SPLINE
SPL {X  -145.877, Y  +737.201, Z    +0.000, E1  +394.468, E3 -267040.191}
SPL {X  -152.550, Y  +719.721, Z    +0.000, E1  +387.728, E3 -267055.680}
SPL {X  -157.145, Y  +701.536, Z    +0.000, E1  +379.368, E3 -267065.135}
SPL {X  -159.035, Y  +688.952, Z    +0.000, E1  +372.676, E3 -267069.176}
SPL {X  -159.756, Y  +680.154, Z    +0.000, E1  +367.520, E3 -267070.903}
SPL {X  -159.986, Y  +672.560, Z    +0.000, E1  +362.636, E3 -267071.801}
SPL {X  -159.990, Y  +668.344, Z    +0.000, E1  +359.382, E3 -267072.067}
SPL {X  -159.990, Y  +664.070, Z    +0.000, E1  +354.975, E3 -267072.395}
SPL {X  -159.990, Y  +656.953, Z    +0.000, E1  +346.040, E3 -267073.462}
SPL {X  -159.990, Y  +644.589, Z    +0.000, E1  +330.989, E3 -267076.873}
SPL {X  -159.990, Y  +605.095, Z    +0.000, E1  +310.486, E3 -267101.964}
SPL {X  -159.990, Y  +546.155, Z    +0.000, E1  +305.539, E3 -267164.723}
SPL {X  -159.990, Y  +539.348, Z    +0.000, E1  +305.531, E3 -267175.026}
SPL {X  -159.990, Y  +530.752, Z    +0.000, E1  +305.518, E3 -267188.034}
SPL {X  -159.990, Y  +522.797, Z    +0.000, E1  +305.537, E3 -267200.117}
SPL {X  -159.990, Y  +515.332, Z    +0.000, E1  +305.526, E3 -267211.406}
SPL {X  -159.990, Y  +508.047, Z    +0.000, E1  +305.531, E3 -267222.422}
SPL {X  -159.990, Y  +501.296, Z    +0.000, E1  +305.518, E3 -267232.644}
SPL {X  -159.990, Y  +487.558, Z    +0.000, E1  +304.151, E3 -267244.274}
SPL {X  -159.990, Y  +454.926, Z    +0.000, E1  +299.433, E3 -267255.714}
SPL {X  -159.990, Y  +449.697, Z    +0.000, E1  +300.191, E3 -267267.176}
SPL {X  -159.990, Y  +445.847, Z    +0.000, E1  +300.905, E3 -267276.799}
SPL {X  -159.990, Y  +439.266, Z    +0.000, E1  +301.568, E3 -267289.882}
SPL {X  -159.990, Y  +432.883, Z    +0.000, E1  +302.386, E3 -267303.573}
SPL {X  -159.990, Y  +429.044, Z    +0.000, E1  +303.109, E3 -267313.463}
SPL {X  -159.990, Y  +425.222, Z    +0.000, E1  +304.101, E3 -267325.360}
SPL {X  -159.990, Y  +418.562, Z    +0.000, E1  +304.950, E3 -267340.518}
SPL {X  -159.990, Y  +407.911, Z    +0.000, E1  +305.062, E3 -267357.109}
SPL {X  -159.990, Y  +400.284, Z    +0.000, E1  +305.103, E3 -267368.543}
SPL {X  -159.990, Y  +391.119, Z    +0.000, E1  +305.052, E3 -267382.131}
SPL {X  -159.988, Y  +381.720, Z    +0.000, E1  +305.103, E3 -267396.239}
SPL {X  -159.786, Y  +374.425, Z    +0.000, E1  +305.121, E3 -267407.287}
SPL {X  -159.015, Y  +364.863, Z    +0.000, E1  +305.220, E3 -267422.303}
SPL {X  -157.966, Y  +357.131, Z    +0.000, E1  +305.441, E3 -267434.993}
SPL {X  -156.775, Y  +350.586, Z    +0.000, E1  +305.627, E3 -267445.967}
SPL {X  -155.027, Y  +342.959, Z    +0.000, E1  +305.926, E3 -267459.140}
SPL {X  -152.882, Y  +335.340, Z    +0.000, E1  +306.305, E3 -267472.683}
SPL {X  -150.681, Y  +328.723, Z    +0.000, E1  +306.710, E3 -267484.777}
SPL {X  -148.661, Y  +323.366, Z    +0.000, E1  +307.100, E3 -267494.786}
SPL {X  -147.089, Y  +319.560, Z    +0.000, E1  +307.396, E3 -267502.002}
SPL {X  -145.161, Y  +315.232, Z    +0.000, E1  +307.745, E3 -267510.282}
SPL {X  -142.534, Y  +309.830, Z    +0.000, E1  +308.237, E3 -267520.787}
SPL {X  -132.342, Y  +292.599, Z    +0.000, E1  +315.826, E3 -267618.075}
ENDSPLINE

SPLINE
SPL {X  -151.238, Y  +330.309, Z    +0.000, E1  +330.693, E3 -267691.232}
SPL {X  -156.949, Y  +351.453, Z    +0.000, E1  +340.161, E3 -267703.393}
SPL {X  -159.024, Y  +364.945, Z    +0.000, E1  +347.297, E3 -267707.811}
SPL {X  -159.758, Y  +373.891, Z    +0.000, E1  +352.513, E3 -267709.699}
SPL {X  -159.985, Y  +381.208, Z    +0.000, E1  +357.184, E3 -267710.582}
SPL {X  -159.990, Y  +384.493, Z    +0.000, E1  +359.676, E3 -267710.807}
SPL {X  -159.990, Y  +387.327, Z    +0.000, E1  +362.137, E3 -267710.990}
SPL {X  -159.990, Y  +392.053, Z    +0.000, E1  +367.477, E3 -267711.454}
SPL {X  -159.990, Y  +396.158, Z    +0.000, E1  +372.775, E3 -267712.080}
SPL {X  -159.990, Y  +401.377, Z    +0.000, E1  +379.398, E3 -267713.260}
SPL {X  -159.990, Y  +411.365, Z    +0.000, E1  +390.630, E3 -267716.469}
SPL {X  -159.990, Y  +450.467, Z    +0.000, E1  +410.183, E3 -267740.118}
SPL {X  -159.990, Y  +509.934, Z    +0.000, E1  +414.923, E3 -267802.736}
SPL {X  -159.990, Y  +516.848, Z    +0.000, E1  +414.930, E3 -267813.025}
SPL {X  -159.990, Y  +524.818, Z    +0.000, E1  +414.933, E3 -267824.896}
SPL {X  -159.990, Y  +532.100, Z    +0.000, E1  +414.924, E3 -267835.749}
SPL {X  -159.990, Y  +539.391, Z    +0.000, E1  +414.933, E3 -267846.601}
SPL {X  -159.990, Y  +546.283, Z    +0.000, E1  +414.924, E3 -267856.873}
SPL {X  -159.990, Y  +553.734, Z    +0.000, E1  +414.938, E3 -267867.960}
SPL {X  -159.990, Y  +564.956, Z    +0.000, E1  +414.973, E3 -267884.631}
SPL {X  -159.990, Y  +577.902, Z    +0.000, E1  +414.969, E3 -267903.921}
SPL {X  -159.990, Y  +588.063, Z    +0.000, E1  +414.931, E3 -267919.112}
SPL {X  -159.990, Y  +595.273, Z    +0.000, E1  +414.928, E3 -267929.835}
SPL {X  -159.990, Y  +602.326, Z    +0.000, E1  +414.932, E3 -267940.336}
SPL {X  -159.990, Y  +609.708, Z    +0.000, E1  +414.930, E3 -267951.342}
SPL {X  -159.990, Y  +618.088, Z    +0.000, E1  +414.948, E3 -267963.771}
SPL {X  -159.990, Y  +625.928, Z    +0.000, E1  +414.931, E3 -267975.467}
SPL {X  -159.990, Y  +632.991, Z    +0.000, E1  +414.938, E3 -267985.970}
SPL {X  -159.990, Y  +639.033, Z    +0.000, E1  +414.931, E3 -267994.978}
SPL {X  -159.990, Y  +646.303, Z    +0.000, E1  +414.946, E3 -268005.766}
SPL {X  -159.990, Y  +656.335, Z    +0.000, E1  +414.969, E3 -268020.668}
SPL {X  -159.990, Y  +664.577, Z    +0.000, E1  +414.924, E3 -268033.045}
SPL {X  -159.989, Y  +672.128, Z    +0.000, E1  +414.946, E3 -268044.262}
SPL {X  -159.636, Y  +682.136, Z    +0.000, E1  +414.901, E3 -268059.520}
SPL {X  -158.805, Y  +690.934, Z    +0.000, E1  +414.742, E3 -268073.531}
SPL {X  -157.890, Y  +697.337, Z    +0.000, E1  +414.571, E3 -268084.052}
SPL {X  -156.492, Y  +704.774, Z    +0.000, E1  +414.365, E3 -268096.531}
SPL {X  -154.917, Y  +711.470, Z    +0.000, E1  +414.052, E3 -268108.191}
SPL {X  -153.204, Y  +717.603, Z    +0.000, E1  +413.775, E3 -268119.037}
SPL {X  -151.355, Y  +723.351, Z    +0.000, E1  +413.415, E3 -268129.508}
SPL {X  -148.967, Y  +729.859, Z    +0.000, E1  +413.026, E3 -268141.520}
SPL {X  -145.862, Y  +737.236, Z    +0.000, E1  +412.427, E3 -268155.575}
SPL {X  -142.777, Y  +743.691, Z    +0.000, E1  +411.831, E3 -268168.118}
SPL {X  -132.301, Y  +761.463, Z    +0.000, E1  +405.510, E3 -268247.403}
ENDSPLINE

SPLINE
SPL {X  -145.877, Y  +737.201, Z    +0.000, E1  +394.468, E3 -268330.514}
SPL {X  -152.550, Y  +719.721, Z    +0.000, E1  +387.728, E3 -268346.003}
SPL {X  -157.145, Y  +701.536, Z    +0.000, E1  +379.368, E3 -268355.458}
SPL {X  -159.035, Y  +688.952, Z    +0.000, E1  +372.676, E3 -268359.499}
SPL {X  -159.756, Y  +680.154, Z    +0.000, E1  +367.520, E3 -268361.225}
SPL {X  -159.986, Y  +672.560, Z    +0.000, E1  +362.636, E3 -268362.123}
SPL {X  -159.990, Y  +668.344, Z    +0.000, E1  +359.382, E3 -268362.389}
SPL {X  -159.990, Y  +664.070, Z    +0.000, E1  +354.975, E3 -268362.718}
SPL {X  -159.990, Y  +656.953, Z    +0.000, E1  +346.040, E3 -268363.784}
SPL {X  -159.990, Y  +644.589, Z    +0.000, E1  +330.989, E3 -268367.196}
SPL {X  -159.990, Y  +605.095, Z    +0.000, E1  +310.486, E3 -268392.287}
SPL {X  -159.990, Y  +546.155, Z    +0.000, E1  +305.539, E3 -268455.045}
SPL {X  -159.990, Y  +539.348, Z    +0.000, E1  +305.531, E3 -268465.349}
SPL {X  -159.990, Y  +530.752, Z    +0.000, E1  +305.518, E3 -268478.356}
SPL {X  -159.990, Y  +522.797, Z    +0.000, E1  +305.537, E3 -268490.439}
SPL {X  -159.990, Y  +515.332, Z    +0.000, E1  +305.526, E3 -268501.728}
SPL {X  -159.990, Y  +508.047, Z    +0.000, E1  +305.531, E3 -268512.745}
SPL {X  -159.990, Y  +501.296, Z    +0.000, E1  +305.518, E3 -268522.966}
SPL {X  -159.990, Y  +487.558, Z    +0.000, E1  +304.151, E3 -268534.597}
SPL {X  -159.990, Y  +454.926, Z    +0.000, E1  +299.433, E3 -268546.036}
SPL {X  -159.990, Y  +449.697, Z    +0.000, E1  +300.191, E3 -268557.499}
SPL {X  -159.990, Y  +445.847, Z    +0.000, E1  +300.905, E3 -268567.122}
SPL {X  -159.990, Y  +439.266, Z    +0.000, E1  +301.568, E3 -268580.205}
SPL {X  -159.990, Y  +432.883, Z    +0.000, E1  +302.386, E3 -268593.895}
SPL {X  -159.990, Y  +428.299, Z    +0.000, E1  +303.316, E3 -268606.299}
SPL {X  -159.990, Y  +424.402, Z    +0.000, E1  +304.297, E3 -268617.974}
SPL {X  -159.990, Y  +420.083, Z    +0.000, E1  +304.918, E3 -268628.258}
SPL {X  -159.990, Y  +412.567, Z    +0.000, E1  +305.072, E3 -268640.482}
SPL {X  -159.990, Y  +405.235, Z    +0.000, E1  +305.098, E3 -268651.471}
SPL {X  -159.990, Y  +400.284, Z    +0.000, E1  +305.103, E3 -268658.865}
SPL {X  -159.990, Y  +391.119, Z    +0.000, E1  +305.052, E3 -268672.454}
SPL {X  -159.988, Y  +381.720, Z    +0.000, E1  +305.103, E3 -268686.561}
SPL {X  -159.786, Y  +374.425, Z    +0.000, E1  +305.121, E3 -268697.609}
SPL {X  -159.015, Y  +364.863, Z    +0.000, E1  +305.220, E3 -268712.626}
SPL {X  -157.966, Y  +357.131, Z    +0.000, E1  +305.441, E3 -268725.316}
SPL {X  -156.775, Y  +350.586, Z    +0.000, E1  +305.627, E3 -268736.290}
SPL {X  -155.397, Y  +344.442, Z    +0.000, E1  +305.886, E3 -268746.906}
SPL {X  -153.976, Y  +339.046, Z    +0.000, E1  +306.128, E3 -268756.398}
SPL {X  -152.417, Y  +333.859, Z    +0.000, E1  +306.416, E3 -268765.724}
SPL {X  -150.681, Y  +328.723, Z    +0.000, E1  +306.710, E3 -268775.100}
SPL {X  -147.884, Y  +321.449, Z    +0.000, E1  +307.200, E3 -268788.673}
SPL {X  -144.518, Y  +313.862, Z    +0.000, E1  +307.832, E3 -268803.219}
SPL {X  -141.812, Y  +308.430, Z    +0.000, E1  +308.410, E3 -268813.906}
SPL {X  -132.342, Y  +292.599, Z    +0.000, E1  +315.826, E3 -268908.398}
ENDSPLINE

SPLINE
SPL {X  -151.238, Y  +330.309, Z    +0.000, E1  +330.693, E3 -268981.554}
SPL {X  -156.949, Y  +351.453, Z    +0.000, E1  +340.161, E3 -268993.715}
SPL {X  -159.024, Y  +364.945, Z    +0.000, E1  +347.297, E3 -268998.133}
SPL {X  -159.878, Y  +376.512, Z    +0.000, E1  +354.071, E3 -269000.385}
SPL {X  -159.990, Y  +382.403, Z    +0.000, E1  +358.090, E3 -269001.004}
SPL {X  -159.990, Y  +385.261, Z    +0.000, E1  +360.259, E3 -269001.175}
SPL {X  -159.990, Y  +389.002, Z    +0.000, E1  +363.890, E3 -269001.453}
SPL {X  -159.990, Y  +394.493, Z    +0.000, E1  +370.512, E3 -269002.128}
SPL {X  -159.990, Y  +401.377, Z    +0.000, E1  +379.398, E3 -269003.583}
SPL {X  -159.990, Y  +411.365, Z    +0.000, E1  +390.630, E3 -269006.791}
SPL {X  -159.990, Y  +450.467, Z    +0.000, E1  +410.183, E3 -269030.440}
SPL {X  -159.990, Y  +509.934, Z    +0.000, E1  +414.923, E3 -269093.059}
SPL {X  -159.990, Y  +516.848, Z    +0.000, E1  +414.930, E3 -269103.347}
SPL {X  -159.990, Y  +524.818, Z    +0.000, E1  +414.933, E3 -269115.219}
SPL {X  -159.990, Y  +532.100, Z    +0.000, E1  +414.924, E3 -269126.072}
SPL {X  -159.990, Y  +539.391, Z    +0.000, E1  +414.933, E3 -269136.924}
SPL {X  -159.990, Y  +546.283, Z    +0.000, E1  +414.924, E3 -269147.196}
SPL {X  -159.990, Y  +553.734, Z    +0.000, E1  +414.938, E3 -269158.282}
SPL {X  -159.990, Y  +564.956, Z    +0.000, E1  +414.973, E3 -269174.954}
SPL {X  -159.990, Y  +577.902, Z    +0.000, E1  +414.969, E3 -269194.243}
SPL {X  -159.990, Y  +588.063, Z    +0.000, E1  +414.931, E3 -269209.434}
SPL {X  -159.990, Y  +595.273, Z    +0.000, E1  +414.928, E3 -269220.158}
SPL {X  -159.990, Y  +602.326, Z    +0.000, E1  +414.932, E3 -269230.658}
SPL {X  -159.990, Y  +609.708, Z    +0.000, E1  +414.930, E3 -269241.665}
SPL {X  -159.990, Y  +618.088, Z    +0.000, E1  +414.948, E3 -269254.094}
SPL {X  -159.990, Y  +625.928, Z    +0.000, E1  +414.931, E3 -269265.790}
SPL {X  -159.990, Y  +635.803, Z    +0.000, E1  +414.980, E3 -269280.418}
SPL {X  -159.990, Y  +646.303, Z    +0.000, E1  +414.946, E3 -269296.088}
SPL {X  -159.990, Y  +653.312, Z    +0.000, E1  +414.932, E3 -269306.540}
SPL {X  -159.990, Y  +658.943, Z    +0.000, E1  +414.931, E3 -269314.938}
SPL {X  -159.990, Y  +667.151, Z    +0.000, E1  +414.954, E3 -269327.157}
SPL {X  -159.885, Y  +677.285, Z    +0.000, E1  +414.936, E3 -269342.352}
SPL {X  -159.482, Y  +684.244, Z    +0.000, E1  +414.840, E3 -269353.204}
SPL {X  -158.805, Y  +690.934, Z    +0.000, E1  +414.742, E3 -269363.853}
SPL {X  -157.890, Y  +697.337, Z    +0.000, E1  +414.571, E3 -269374.375}
SPL {X  -156.492, Y  +704.774, Z    +0.000, E1  +414.365, E3 -269386.854}
SPL {X  -154.917, Y  +711.470, Z    +0.000, E1  +414.052, E3 -269398.514}
SPL {X  -153.204, Y  +717.603, Z    +0.000, E1  +413.775, E3 -269409.360}
SPL {X  -151.355, Y  +723.351, Z    +0.000, E1  +413.415, E3 -269419.831}
SPL {X  -148.967, Y  +729.859, Z    +0.000, E1  +413.026, E3 -269431.843}
SPL {X  -145.862, Y  +737.236, Z    +0.000, E1  +412.427, E3 -269445.897}
SPL {X  -142.777, Y  +743.691, Z    +0.000, E1  +411.831, E3 -269458.441}
SPL {X  -132.301, Y  +761.463, Z    +0.000, E1  +405.510, E3 -269537.726}
ENDSPLINE

SPLINE
SPL {X  -145.877, Y  +737.201, Z    +0.000, E1  +394.468, E3 -269620.836}
SPL {X  -152.550, Y  +719.721, Z    +0.000, E1  +387.728, E3 -269636.326}
SPL {X  -157.145, Y  +701.536, Z    +0.000, E1  +379.368, E3 -269645.780}
SPL {X  -159.035, Y  +688.952, Z    +0.000, E1  +372.676, E3 -269649.821}
SPL {X  -159.873, Y  +677.622, Z    +0.000, E1  +366.008, E3 -269651.893}
SPL {X  -159.990, Y  +670.381, Z    +0.000, E1  +361.064, E3 -269652.594}
SPL {X  -159.990, Y  +666.603, Z    +0.000, E1  +357.744, E3 -269652.825}
SPL {X  -159.990, Y  +661.750, Z    +0.000, E1  +352.120, E3 -269653.298}
SPL {X  -159.990, Y  +657.656, Z    +0.000, E1  +346.724, E3 -269653.943}
SPL {X  -159.990, Y  +652.023, Z    +0.000, E1  +339.551, E3 -269655.231}
SPL {X  -159.990, Y  +641.935, Z    +0.000, E1  +328.152, E3 -269658.403}
SPL {X  -159.990, Y  +605.095, Z    +0.000, E1  +310.486, E3 -269682.609}
SPL {X  -159.990, Y  +546.155, Z    +0.000, E1  +305.539, E3 -269745.368}
SPL {X  -159.990, Y  +539.348, Z    +0.000, E1  +305.531, E3 -269755.672}
SPL {X  -159.990, Y  +530.752, Z    +0.000, E1  +305.518, E3 -269768.679}
SPL {X  -159.990, Y  +522.797, Z    +0.000, E1  +305.537, E3 -269780.762}
SPL {X  -159.990, Y  +515.332, Z    +0.000, E1  +305.526, E3 -269792.051}
SPL {X  -159.990, Y  +508.047, Z    +0.000, E1  +305.531, E3 -269803.068}
SPL {X  -159.990, Y  +499.403, Z    +0.000, E1  +305.488, E3 -269816.107}
SPL {X  -159.990, Y  +479.413, Z    +0.000, E1  +302.719, E3 -269827.252}
SPL {X  -159.990, Y  +454.926, Z    +0.000, E1  +299.433, E3 -269836.359}
SPL {X  -159.990, Y  +449.697, Z    +0.000, E1  +300.191, E3 -269847.821}
SPL {X  -159.990, Y  +445.847, Z    +0.000, E1  +300.905, E3 -269857.444}
SPL {X  -159.990, Y  +439.266, Z    +0.000, E1  +301.568, E3 -269870.528}
SPL {X  -159.990, Y  +432.883, Z    +0.000, E1  +302.386, E3 -269884.218}
SPL {X  -159.990, Y  +428.299, Z    +0.000, E1  +303.316, E3 -269896.621}
SPL {X  -159.990, Y  +424.402, Z    +0.000, E1  +304.297, E3 -269908.296}
SPL {X  -159.990, Y  +418.562, Z    +0.000, E1  +304.950, E3 -269921.163}
SPL {X  -159.990, Y  +410.722, Z    +0.000, E1  +305.100, E3 -269933.624}
SPL {X  -159.990, Y  +402.790, Z    +0.000, E1  +305.070, E3 -269945.399}
SPL {X  -159.990, Y  +392.953, Z    +0.000, E1  +305.082, E3 -269960.093}
SPL {X  -159.990, Y  +383.354, Z    +0.000, E1  +305.080, E3 -269974.403}
SPL {X  -159.786, Y  +374.425, Z    +0.000, E1  +305.121, E3 -269987.932}
SPL {X  -159.015, Y  +364.863, Z    +0.000, E1  +305.220, E3 -270002.948}
SPL {X  -157.966, Y  +357.131, Z    +0.000, E1  +305.441, E3 -270015.639}
SPL {X  -156.775, Y  +350.586, Z    +0.000, E1  +305.627, E3 -270026.613}
SPL {X  -155.027, Y  +342.959, Z    +0.000, E1  +305.926, E3 -270039.786}
SPL {X  -152.882, Y  +335.340, Z    +0.000, E1  +306.305, E3 -270053.328}
SPL {X  -150.681, Y  +328.723, Z    +0.000, E1  +306.710, E3 -270065.422}
SPL {X  -147.884, Y  +321.449, Z    +0.000, E1  +307.200, E3 -270078.996}
SPL {X  -145.161, Y  +315.232, Z    +0.000, E1  +307.745, E3 -270090.927}
SPL {X  -142.534, Y  +309.830, Z    +0.000, E1  +308.237, E3 -270101.432}
SPL {X  -132.342, Y  +292.599, Z    +0.000, E1  +315.826, E3 -270198.720}
ENDSPLINE

SPLINE
SPL {X  -151.238, Y  +330.309, Z    +0.000, E1  +330.693, E3 -270271.877}
SPL {X  -156.949, Y  +351.453, Z    +0.000, E1  +340.161, E3 -270284.038}
SPL {X  -159.024, Y  +364.945, Z    +0.000, E1  +347.297, E3 -270288.456}
SPL {X  -159.758, Y  +373.891, Z    +0.000, E1  +352.513, E3 -270290.344}
SPL {X  -159.985, Y  +381.208, Z    +0.000, E1  +357.184, E3 -270291.227}
SPL {X  -159.990, Y  +385.261, Z    +0.000, E1  +360.259, E3 -270291.497}
SPL {X  -159.990, Y  +388.094, Z    +0.000, E1  +363.012, E3 -270291.690}
SPL {X  -159.990, Y  +392.053, Z    +0.000, E1  +367.477, E3 -270292.100}
SPL {X  -159.990, Y  +396.158, Z    +0.000, E1  +372.775, E3 -270292.725}
SPL {X  -159.990, Y  +401.377, Z    +0.000, E1  +379.398, E3 -270293.905}
SPL {X  -159.990, Y  +411.365, Z    +0.000, E1  +390.630, E3 -270297.114}
SPL {X  -159.990, Y  +450.467, Z    +0.000, E1  +410.183, E3 -270320.763}
SPL {X  -159.990, Y  +509.934, Z    +0.000, E1  +414.923, E3 -270383.382}
SPL {X  -159.990, Y  +516.848, Z    +0.000, E1  +414.930, E3 -270393.670}
SPL {X  -159.990, Y  +524.818, Z    +0.000, E1  +414.933, E3 -270405.542}
SPL {X  -159.990, Y  +532.100, Z    +0.000, E1  +414.924, E3 -270416.395}
SPL {X  -159.990, Y  +539.391, Z    +0.000, E1  +414.933, E3 -270427.247}
SPL {X  -159.990, Y  +546.283, Z    +0.000, E1  +414.924, E3 -270437.518}
SPL {X  -159.990, Y  +553.734, Z    +0.000, E1  +414.938, E3 -270448.605}
SPL {X  -159.990, Y  +560.657, Z    +0.000, E1  +414.914, E3 -270458.966}
SPL {X  -159.990, Y  +567.311, Z    +0.000, E1  +414.931, E3 -270468.851}
SPL {X  -159.990, Y  +577.902, Z    +0.000, E1  +414.969, E3 -270484.566}
SPL {X  -159.990, Y  +588.063, Z    +0.000, E1  +414.931, E3 -270499.757}
SPL {X  -159.990, Y  +595.273, Z    +0.000, E1  +414.928, E3 -270510.480}
SPL {X  -159.990, Y  +602.326, Z    +0.000, E1  +414.932, E3 -270520.981}
SPL {X  -159.990, Y  +609.708, Z    +0.000, E1  +414.930, E3 -270531.988}
SPL {X  -159.990, Y  +618.088, Z    +0.000, E1  +414.948, E3 -270544.416}
SPL {X  -159.990, Y  +625.928, Z    +0.000, E1  +414.931, E3 -270556.112}
SPL {X  -159.990, Y  +635.803, Z    +0.000, E1  +414.980, E3 -270570.740}
SPL {X  -159.990, Y  +646.303, Z    +0.000, E1  +414.946, E3 -270586.411}
SPL {X  -159.990, Y  +653.312, Z    +0.000, E1  +414.932, E3 -270596.863}
SPL {X  -159.990, Y  +658.943, Z    +0.000, E1  +414.931, E3 -270605.261}
SPL {X  -159.990, Y  +667.151, Z    +0.000, E1  +414.954, E3 -270617.479}
SPL {X  -159.885, Y  +677.285, Z    +0.000, E1  +414.936, E3 -270632.675}
SPL {X  -159.482, Y  +684.244, Z    +0.000, E1  +414.840, E3 -270643.527}
SPL {X  -158.805, Y  +690.934, Z    +0.000, E1  +414.742, E3 -270654.176}
SPL {X  -157.890, Y  +697.337, Z    +0.000, E1  +414.571, E3 -270664.697}
SPL {X  -156.492, Y  +704.774, Z    +0.000, E1  +414.365, E3 -270677.176}
SPL {X  -154.917, Y  +711.470, Z    +0.000, E1  +414.052, E3 -270688.836}
SPL {X  -153.204, Y  +717.603, Z    +0.000, E1  +413.775, E3 -270699.682}
SPL {X  -151.355, Y  +723.351, Z    +0.000, E1  +413.415, E3 -270710.154}
SPL {X  -149.700, Y  +727.952, Z    +0.000, E1  +413.118, E3 -270718.648}
SPL {X  -147.376, Y  +733.767, Z    +0.000, E1  +412.706, E3 -270729.598}
SPL {X  -144.332, Y  +740.529, Z    +0.000, E1  +412.133, E3 -270742.588}
SPL {X  -142.065, Y  +745.081, Z    +0.000, E1  +411.654, E3 -270751.541}
SPL {X  -132.301, Y  +761.463, Z    +0.000, E1  +405.510, E3 -270828.048}
ENDSPLINE

SPLINE
SPL {X  -145.877, Y  +737.201, Z    +0.000, E1  +394.468, E3 -270911.159}
SPL {X  -152.550, Y  +719.721, Z    +0.000, E1  +387.728, E3 -270926.648}
SPL {X  -157.145, Y  +701.536, Z    +0.000, E1  +379.368, E3 -270936.103}
SPL {X  -159.035, Y  +688.952, Z    +0.000, E1  +372.676, E3 -270940.144}
SPL {X  -159.756, Y  +680.154, Z    +0.000, E1  +367.520, E3 -270941.870}
SPL {X  -159.986, Y  +672.560, Z    +0.000, E1  +362.636, E3 -270942.768}
SPL {X  -159.990, Y  +668.344, Z    +0.000, E1  +359.382, E3 -270943.035}
SPL {X  -159.990, Y  +664.070, Z    +0.000, E1  +354.975, E3 -270943.363}
SPL {X  -159.990, Y  +656.953, Z    +0.000, E1  +346.040, E3 -270944.429}
SPL {X  -159.990, Y  +644.589, Z    +0.000, E1  +330.989, E3 -270947.841}
SPL {X  -159.990, Y  +605.095, Z    +0.000, E1  +310.486, E3 -270972.932}
SPL {X  -159.990, Y  +546.155, Z    +0.000, E1  +305.539, E3 -271035.690}
SPL {X  -159.990, Y  +539.348, Z    +0.000, E1  +305.531, E3 -271045.994}
SPL {X  -159.990, Y  +530.752, Z    +0.000, E1  +305.518, E3 -271059.002}
SPL {X  -159.990, Y  +522.797, Z    +0.000, E1  +305.537, E3 -271071.085}
SPL {X  -159.990, Y  +515.332, Z    +0.000, E1  +305.526, E3 -271082.373}
SPL {X  -159.990, Y  +508.047, Z    +0.000, E1  +305.531, E3 -271093.390}
SPL {X  -159.990, Y  +501.296, Z    +0.000, E1  +305.518, E3 -271103.612}
SPL {X  -159.990, Y  +487.558, Z    +0.000, E1  +304.151, E3 -271115.242}
SPL {X  -159.990, Y  +454.926, Z    +0.000, E1  +299.433, E3 -271126.681}
SPL {X  -159.990, Y  +449.697, Z    +0.000, E1  +300.191, E3 -271138.144}
SPL {X  -159.990, Y  +444.026, Z    +0.000, E1  +301.072, E3 -271151.402}
SPL {X  -159.990, Y  +437.596, Z    +0.000, E1  +301.764, E3 -271164.144}
SPL {X  -159.990, Y  +432.883, Z    +0.000, E1  +302.386, E3 -271174.540}
SPL {X  -159.990, Y  +429.044, Z    +0.000, E1  +303.109, E3 -271184.431}
SPL {X  -159.990, Y  +425.222, Z    +0.000, E1  +304.101, E3 -271196.328}
SPL {X  -159.990, Y  +418.562, Z    +0.000, E1  +304.950, E3 -271211.485}
SPL {X  -159.990, Y  +407.911, Z    +0.000, E1  +305.062, E3 -271228.077}
SPL {X  -159.990, Y  +400.284, Z    +0.000, E1  +305.103, E3 -271239.511}
SPL {X  -159.990, Y  +392.953, Z    +0.000, E1  +305.082, E3 -271250.415}
SPL {X  -159.990, Y  +383.354, Z    +0.000, E1  +305.080, E3 -271264.725}
SPL {X  -159.786, Y  +374.425, Z    +0.000, E1  +305.121, E3 -271278.255}
SPL {X  -159.184, Y  +366.462, Z    +0.000, E1  +305.220, E3 -271290.755}
SPL {X  -158.166, Y  +358.413, Z    +0.000, E1  +305.386, E3 -271303.811}
SPL {X  -156.775, Y  +350.586, Z    +0.000, E1  +305.627, E3 -271316.935}
SPL {X  -155.397, Y  +344.442, Z    +0.000, E1  +305.886, E3 -271327.551}
SPL {X  -153.976, Y  +339.046, Z    +0.000, E1  +306.128, E3 -271337.043}
SPL {X  -152.417, Y  +333.859, Z    +0.000, E1  +306.416, E3 -271346.369}
SPL {X  -150.681, Y  +328.723, Z    +0.000, E1  +306.710, E3 -271355.745}
SPL {X  -147.884, Y  +321.449, Z    +0.000, E1  +307.200, E3 -271369.318}
SPL {X  -145.161, Y  +315.232, Z    +0.000, E1  +307.745, E3 -271381.250}
SPL {X  -142.534, Y  +309.830, Z    +0.000, E1  +308.237, E3 -271391.755}
SPL {X  -132.342, Y  +292.599, Z    +0.000, E1  +315.826, E3 -271489.043}
ENDSPLINE

SPLINE
SPL {X  -151.238, Y  +330.309, Z    +0.000, E1  +330.693, E3 -271562.200}
SPL {X  -156.949, Y  +351.453, Z    +0.000, E1  +340.161, E3 -271574.361}
SPL {X  -159.024, Y  +364.945, Z    +0.000, E1  +347.297, E3 -271578.778}
SPL {X  -159.878, Y  +376.512, Z    +0.000, E1  +354.071, E3 -271581.030}
SPL {X  -159.990, Y  +383.659, Z    +0.000, E1  +358.950, E3 -271581.724}
SPL {X  -159.990, Y  +387.327, Z    +0.000, E1  +362.137, E3 -271581.957}
SPL {X  -159.990, Y  +392.053, Z    +0.000, E1  +367.477, E3 -271582.422}
SPL {X  -159.990, Y  +396.158, Z    +0.000, E1  +372.775, E3 -271583.048}
SPL {X  -159.990, Y  +401.377, Z    +0.000, E1  +379.398, E3 -271584.228}
SPL {X  -159.990, Y  +411.365, Z    +0.000, E1  +390.630, E3 -271587.437}
SPL {X  -159.990, Y  +450.467, Z    +0.000, E1  +410.183, E3 -271611.085}
SPL {X  -159.990, Y  +509.934, Z    +0.000, E1  +414.923, E3 -271673.704}
SPL {X  -159.990, Y  +516.848, Z    +0.000, E1  +414.930, E3 -271683.992}
SPL {X  -159.990, Y  +524.818, Z    +0.000, E1  +414.933, E3 -271695.864}
SPL {X  -159.990, Y  +532.100, Z    +0.000, E1  +414.924, E3 -271706.717}
SPL {X  -159.990, Y  +539.391, Z    +0.000, E1  +414.933, E3 -271717.569}
SPL {X  -159.990, Y  +546.283, Z    +0.000, E1  +414.924, E3 -271727.841}
SPL {X  -159.990, Y  +553.734, Z    +0.000, E1  +414.938, E3 -271738.928}
SPL {X  -159.990, Y  +564.956, Z    +0.000, E1  +414.973, E3 -271755.599}
SPL {X  -159.990, Y  +577.902, Z    +0.000, E1  +414.969, E3 -271774.889}
SPL {X  -159.990, Y  +588.063, Z    +0.000, E1  +414.931, E3 -271790.080}
SPL {X  -159.990, Y  +595.273, Z    +0.000, E1  +414.928, E3 -271800.803}
SPL {X  -159.990, Y  +602.326, Z    +0.000, E1  +414.932, E3 -271811.303}
SPL {X  -159.990, Y  +609.708, Z    +0.000, E1  +414.930, E3 -271822.310}
SPL {X  -159.990, Y  +616.306, Z    +0.000, E1  +414.927, E3 -271832.124}
SPL {X  -159.990, Y  +624.320, Z    +0.000, E1  +414.952, E3 -271844.007}
SPL {X  -159.990, Y  +632.991, Z    +0.000, E1  +414.938, E3 -271856.938}
SPL {X  -159.990, Y  +639.033, Z    +0.000, E1  +414.931, E3 -271865.946}
SPL {X  -159.990, Y  +646.303, Z    +0.000, E1  +414.946, E3 -271876.733}
SPL {X  -159.990, Y  +656.335, Z    +0.000, E1  +414.969, E3 -271891.636}
SPL {X  -159.990, Y  +664.577, Z    +0.000, E1  +414.924, E3 -271904.013}
SPL {X  -159.989, Y  +672.128, Z    +0.000, E1  +414.946, E3 -271915.230}
SPL {X  -159.792, Y  +679.466, Z    +0.000, E1  +414.893, E3 -271926.388}
SPL {X  -159.330, Y  +686.016, Z    +0.000, E1  +414.837, E3 -271936.619}
SPL {X  -158.190, Y  +695.432, Z    +0.000, E1  +414.658, E3 -271951.815}
SPL {X  -157.027, Y  +702.151, Z    +0.000, E1  +414.415, E3 -271963.097}
SPL {X  -156.112, Y  +706.513, Z    +0.000, E1  +414.265, E3 -271970.531}
SPL {X  -154.917, Y  +711.470, Z    +0.000, E1  +414.052, E3 -271979.159}
SPL {X  -153.561, Y  +716.398, Z    +0.000, E1  +413.816, E3 -271987.880}
SPL {X  -151.715, Y  +722.287, Z    +0.000, E1  +413.503, E3 -271998.496}
SPL {X  -148.967, Y  +729.859, Z    +0.000, E1  +413.026, E3 -272012.488}
SPL {X  -146.734, Y  +735.264, Z    +0.000, E1  +412.550, E3 -272022.820}
SPL {X  -144.332, Y  +740.529, Z    +0.000, E1  +412.133, E3 -272032.911}
SPL {X  -142.065, Y  +745.081, Z    +0.000, E1  +411.654, E3 -272041.864}
SPL {X  -132.301, Y  +761.463, Z    +0.000, E1  +405.510, E3 -272118.371}
ENDSPLINE

SPLINE
SPL {X  -145.877, Y  +737.201, Z    +0.000, E1  +394.468, E3 -272201.482}
SPL {X  -152.550, Y  +719.721, Z    +0.000, E1  +387.728, E3 -272216.971}
SPL {X  -157.145, Y  +701.536, Z    +0.000, E1  +379.368, E3 -272226.425}
SPL {X  -159.035, Y  +688.952, Z    +0.000, E1  +372.676, E3 -272230.466}
SPL {X  -159.873, Y  +677.622, Z    +0.000, E1  +366.008, E3 -272232.538}
SPL {X  -159.990, Y  +670.381, Z    +0.000, E1  +361.064, E3 -272233.239}
SPL {X  -159.990, Y  +667.647, Z    +0.000, E1  +358.660, E3 -272233.397}
SPL {X  -159.990, Y  +664.070, Z    +0.000, E1  +354.975, E3 -272233.685}
SPL {X  -159.990, Y  +658.737, Z    +0.000, E1  +348.199, E3 -272234.392}
SPL {X  -159.990, Y  +652.023, Z    +0.000, E1  +339.551, E3 -272235.876}
SPL {X  -159.990, Y  +641.935, Z    +0.000, E1  +328.152, E3 -272239.048}
SPL {X  -159.990, Y  +605.095, Z    +0.000, E1  +310.486, E3 -272263.254}
SPL {X  -159.990, Y  +546.155, Z    +0.000, E1  +305.539, E3 -272326.013}
SPL {X  -159.990, Y  +539.348, Z    +0.000, E1  +305.531, E3 -272336.317}
SPL {X  -159.990, Y  +530.752, Z    +0.000, E1  +305.518, E3 -272349.324}
SPL {X  -159.990, Y  +522.797, Z    +0.000, E1  +305.537, E3 -272361.407}
SPL {X  -159.990, Y  +515.332, Z    +0.000, E1  +305.526, E3 -272372.696}
SPL {X  -159.990, Y  +508.047, Z    +0.000, E1  +305.531, E3 -272383.713}
SPL {X  -159.990, Y  +499.403, Z    +0.000, E1  +305.488, E3 -272396.752}
SPL {X  -159.990, Y  +479.413, Z    +0.000, E1  +302.719, E3 -272407.897}
SPL {X  -159.990, Y  +454.926, Z    +0.000, E1  +299.433, E3 -272417.004}
SPL {X  -159.990, Y  +449.697, Z    +0.000, E1  +300.191, E3 -272428.466}
SPL {X  -159.990, Y  +444.026, Z    +0.000, E1  +301.072, E3 -272441.725}
SPL {X  -159.990, Y  +437.596, Z    +0.000, E1  +301.764, E3 -272454.466}
SPL {X  -159.990, Y  +432.883, Z    +0.000, E1  +302.386, E3 -272464.863}
SPL {X  -159.990, Y  +429.044, Z    +0.000, E1  +303.109, E3 -272474.753}
SPL {X  -159.990, Y  +425.222, Z    +0.000, E1  +304.101, E3 -272486.650}
SPL {X  -159.990, Y  +418.562, Z    +0.000, E1  +304.950, E3 -272501.808}
SPL {X  -159.990, Y  +410.722, Z    +0.000, E1  +305.100, E3 -272514.269}
SPL {X  -159.990, Y  +402.790, Z    +0.000, E1  +305.070, E3 -272526.044}
SPL {X  -159.990, Y  +391.119, Z    +0.000, E1  +305.052, E3 -272543.422}
SPL {X  -159.988, Y  +381.720, Z    +0.000, E1  +305.103, E3 -272557.529}
SPL {X  -159.786, Y  +374.425, Z    +0.000, E1  +305.121, E3 -272568.577}
SPL {X  -159.015, Y  +364.863, Z    +0.000, E1  +305.220, E3 -272583.593}
SPL {X  -157.966, Y  +357.131, Z    +0.000, E1  +305.441, E3 -272596.284}
SPL {X  -156.775, Y  +350.586, Z    +0.000, E1  +305.627, E3 -272607.258}
SPL {X  -155.397, Y  +344.442, Z    +0.000, E1  +305.886, E3 -272617.873}
SPL {X  -153.976, Y  +339.046, Z    +0.000, E1  +306.128, E3 -272627.366}
SPL {X  -152.417, Y  +333.859, Z    +0.000, E1  +306.416, E3 -272636.692}
SPL {X  -150.681, Y  +328.723, Z    +0.000, E1  +306.710, E3 -272646.068}
SPL {X  -147.884, Y  +321.449, Z    +0.000, E1  +307.200, E3 -272659.641}
SPL {X  -145.161, Y  +315.232, Z    +0.000, E1  +307.745, E3 -272671.572}
SPL {X  -142.534, Y  +309.830, Z    +0.000, E1  +308.237, E3 -272682.077}
SPL {X  -132.342, Y  +292.599, Z    +0.000, E1  +315.826, E3 -272779.366}
ENDSPLINE

SPLINE
SPL {X  -151.238, Y  +330.309, Z    +0.000, E1  +330.693, E3 -272852.522}
SPL {X  -156.949, Y  +351.453, Z    +0.000, E1  +340.161, E3 -272864.683}
SPL {X  -159.024, Y  +364.945, Z    +0.000, E1  +347.297, E3 -272869.101}
SPL {X  -159.758, Y  +373.891, Z    +0.000, E1  +352.513, E3 -272870.990}
SPL {X  -159.985, Y  +381.208, Z    +0.000, E1  +357.184, E3 -272871.872}
SPL {X  -159.990, Y  +384.493, Z    +0.000, E1  +359.676, E3 -272872.097}
SPL {X  -159.990, Y  +387.327, Z    +0.000, E1  +362.137, E3 -272872.280}
SPL {X  -159.990, Y  +392.053, Z    +0.000, E1  +367.477, E3 -272872.745}
SPL {X  -159.990, Y  +396.158, Z    +0.000, E1  +372.775, E3 -272873.370}
SPL {X  -159.990, Y  +401.377, Z    +0.000, E1  +379.398, E3 -272874.551}
SPL {X  -159.990, Y  +411.365, Z    +0.000, E1  +390.630, E3 -272877.759}
SPL {X  -159.990, Y  +450.467, Z    +0.000, E1  +410.183, E3 -272901.408}
SPL {X  -159.990, Y  +509.934, Z    +0.000, E1  +414.923, E3 -272964.027}
SPL {X  -159.990, Y  +516.848, Z    +0.000, E1  +414.930, E3 -272974.315}
SPL {X  -159.990, Y  +524.818, Z    +0.000, E1  +414.933, E3 -272986.187}
SPL {X  -159.990, Y  +532.100, Z    +0.000, E1  +414.924, E3 -272997.040}
SPL {X  -159.990, Y  +539.391, Z    +0.000, E1  +414.933, E3 -273007.892}
SPL {X  -159.990, Y  +546.283, Z    +0.000, E1  +414.924, E3 -273018.163}
SPL {X  -159.990, Y  +553.734, Z    +0.000, E1  +414.938, E3 -273029.250}
SPL {X  -159.990, Y  +564.956, Z    +0.000, E1  +414.973, E3 -273045.921}
SPL {X  -159.990, Y  +577.902, Z    +0.000, E1  +414.969, E3 -273065.211}
SPL {X  -159.990, Y  +588.063, Z    +0.000, E1  +414.931, E3 -273080.402}
SPL {X  -159.990, Y  +595.273, Z    +0.000, E1  +414.928, E3 -273091.126}
SPL {X  -159.990, Y  +602.326, Z    +0.000, E1  +414.932, E3 -273101.626}
SPL {X  -159.990, Y  +609.708, Z    +0.000, E1  +414.930, E3 -273112.633}
SPL {X  -159.990, Y  +618.088, Z    +0.000, E1  +414.948, E3 -273125.062}
SPL {X  -159.990, Y  +625.928, Z    +0.000, E1  +414.931, E3 -273136.758}
SPL {X  -159.990, Y  +635.803, Z    +0.000, E1  +414.980, E3 -273151.386}
SPL {X  -159.990, Y  +646.303, Z    +0.000, E1  +414.946, E3 -273167.056}
SPL {X  -159.990, Y  +653.312, Z    +0.000, E1  +414.932, E3 -273177.508}
SPL {X  -159.990, Y  +661.828, Z    +0.000, E1  +414.965, E3 -273190.164}
SPL {X  -159.989, Y  +672.128, Z    +0.000, E1  +414.946, E3 -273205.552}
SPL {X  -159.636, Y  +682.136, Z    +0.000, E1  +414.901, E3 -273220.811}
SPL {X  -158.805, Y  +690.934, Z    +0.000, E1  +414.742, E3 -273234.821}
SPL {X  -157.512, Y  +699.550, Z    +0.000, E1  +414.543, E3 -273248.972}
SPL {X  -156.112, Y  +706.513, Z    +0.000, E1  +414.265, E3 -273260.854}
SPL {X  -154.917, Y  +711.470, Z    +0.000, E1  +414.052, E3 -273269.481}
SPL {X  -153.561, Y  +716.398, Z    +0.000, E1  +413.816, E3 -273278.203}
SPL {X  -151.715, Y  +722.287, Z    +0.000, E1  +413.503, E3 -273288.819}
SPL {X  -149.700, Y  +727.952, Z    +0.000, E1  +413.118, E3 -273299.293}
SPL {X  -147.376, Y  +733.767, Z    +0.000, E1  +412.706, E3 -273310.243}
SPL {X  -145.109, Y  +738.881, Z    +0.000, E1  +412.243, E3 -273320.090}
SPL {X  -142.777, Y  +743.691, Z    +0.000, E1  +411.831, E3 -273329.408}
SPL {X  -132.301, Y  +761.463, Z    +0.000, E1  +405.510, E3 -273408.693}
ENDSPLINE

SPLINE
SPL {X  -145.877, Y  +737.201, Z    +0.000, E1  +394.468, E3 -273491.804}
SPL {X  -152.550, Y  +719.721, Z    +0.000, E1  +387.728, E3 -273507.293}
SPL {X  -157.145, Y  +701.536, Z    +0.000, E1  +379.368, E3 -273516.748}
SPL {X  -159.035, Y  +688.952, Z    +0.000, E1  +372.676, E3 -273520.789}
SPL {X  -159.756, Y  +680.154, Z    +0.000, E1  +367.520, E3 -273522.515}
SPL {X  -159.986, Y  +672.560, Z    +0.000, E1  +362.636, E3 -273523.414}
SPL {X  -159.990, Y  +668.344, Z    +0.000, E1  +359.382, E3 -273523.680}
SPL {X  -159.990, Y  +664.070, Z    +0.000, E1  +354.975, E3 -273524.008}
SPL {X  -159.990, Y  +656.953, Z    +0.000, E1  +346.040, E3 -273525.075}
SPL {X  -159.990, Y  +644.589, Z    +0.000, E1  +330.989, E3 -273528.486}
SPL {X  -159.990, Y  +605.095, Z    +0.000, E1  +310.486, E3 -273553.577}
SPL {X  -159.990, Y  +546.155, Z    +0.000, E1  +305.539, E3 -273616.336}
SPL {X  -159.990, Y  +539.348, Z    +0.000, E1  +305.531, E3 -273626.639}
SPL {X  -159.990, Y  +530.752, Z    +0.000, E1  +305.518, E3 -273639.647}
SPL {X  -159.990, Y  +522.797, Z    +0.000, E1  +305.537, E3 -273651.730}
SPL {X  -159.990, Y  +515.332, Z    +0.000, E1  +305.526, E3 -273663.019}
SPL {X  -159.990, Y  +508.047, Z    +0.000, E1  +305.531, E3 -273674.035}
SPL {X  -159.990, Y  +501.296, Z    +0.000, E1  +305.518, E3 -273684.257}
SPL {X  -159.990, Y  +487.558, Z    +0.000, E1  +304.151, E3 -273695.887}
SPL {X  -159.990, Y  +454.926, Z    +0.000, E1  +299.433, E3 -273707.326}
SPL {X  -159.990, Y  +449.697, Z    +0.000, E1  +300.191, E3 -273718.789}
SPL {X  -159.990, Y  +445.847, Z    +0.000, E1  +300.905, E3 -273728.412}
SPL {X  -159.990, Y  +439.266, Z    +0.000, E1  +301.568, E3 -273741.495}
SPL {X  -159.990, Y  +432.883, Z    +0.000, E1  +302.386, E3 -273755.186}
SPL {X  -159.990, Y  +429.044, Z    +0.000, E1  +303.109, E3 -273765.076}
SPL {X  -159.990, Y  +425.222, Z    +0.000, E1  +304.101, E3 -273776.973}
SPL {X  -159.990, Y  +420.083, Z    +0.000, E1  +304.918, E3 -273789.549}
SPL {X  -159.990, Y  +412.567, Z    +0.000, E1  +305.072, E3 -273801.773}
SPL {X  -159.990, Y  +405.235, Z    +0.000, E1  +305.098, E3 -273812.761}
SPL {X  -159.990, Y  +400.284, Z    +0.000, E1  +305.103, E3 -273820.156}
SPL {X  -159.990, Y  +391.119, Z    +0.000, E1  +305.052, E3 -273833.744}
SPL {X  -159.988, Y  +381.720, Z    +0.000, E1  +305.103, E3 -273847.852}
SPL {X  -159.786, Y  +374.425, Z    +0.000, E1  +305.121, E3 -273858.900}
SPL {X  -159.184, Y  +366.462, Z    +0.000, E1  +305.220, E3 -273871.400}
SPL {X  -158.166, Y  +358.413, Z    +0.000, E1  +305.386, E3 -273884.456}
SPL {X  -156.775, Y  +350.586, Z    +0.000, E1  +305.627, E3 -273897.580}
SPL {X  -155.027, Y  +342.959, Z    +0.000, E1  +305.926, E3 -273910.753}
SPL {X  -152.882, Y  +335.340, Z    +0.000, E1  +306.305, E3 -273924.296}
SPL {X  -150.681, Y  +328.723, Z    +0.000, E1  +306.710, E3 -273936.390}
SPL {X  -147.884, Y  +321.449, Z    +0.000, E1  +307.200, E3 -273949.963}
SPL {X  -144.518, Y  +313.862, Z    +0.000, E1  +307.832, E3 -273964.509}
SPL {X  -141.812, Y  +308.430, Z    +0.000, E1  +308.410, E3 -273975.197}
SPL {X  -132.342, Y  +292.599, Z    +0.000, E1  +315.826, E3 -274069.688}
ENDSPLINE

SPLINE
SPL {X  -151.238, Y  +330.309, Z    +0.000, E1  +330.693, E3 -274142.845}
SPL {X  -156.949, Y  +351.453, Z    +0.000, E1  +340.161, E3 -274155.006}
SPL {X  -159.024, Y  +364.945, Z    +0.000, E1  +347.297, E3 -274159.423}
SPL {X  -159.758, Y  +373.891, Z    +0.000, E1  +352.513, E3 -274161.312}
SPL {X  -159.985, Y  +381.208, Z    +0.000, E1  +357.184, E3 -274162.195}
SPL {X  -159.990, Y  +384.493, Z    +0.000, E1  +359.676, E3 -274162.420}
SPL {X  -159.990, Y  +387.327, Z    +0.000, E1  +362.137, E3 -274162.602}
SPL {X  -159.990, Y  +392.053, Z    +0.000, E1  +367.477, E3 -274163.067}
SPL {X  -159.990, Y  +396.158, Z    +0.000, E1  +372.775, E3 -274163.693}
SPL {X  -159.990, Y  +401.377, Z    +0.000, E1  +379.398, E3 -274164.873}
SPL {X  -159.990, Y  +411.365, Z    +0.000, E1  +390.630, E3 -274168.082}
SPL {X  -159.990, Y  +450.467, Z    +0.000, E1  +410.183, E3 -274191.731}
SPL {X  -159.990, Y  +509.934, Z    +0.000, E1  +414.923, E3 -274254.349}
SPL {X  -159.990, Y  +516.848, Z    +0.000, E1  +414.930, E3 -274264.637}
SPL {X  -159.990, Y  +524.818, Z    +0.000, E1  +414.933, E3 -274276.509}
SPL {X  -159.990, Y  +532.100, Z    +0.000, E1  +414.924, E3 -274287.362}
SPL {X  -159.990, Y  +539.391, Z    +0.000, E1  +414.933, E3 -274298.214}
SPL {X  -159.990, Y  +546.283, Z    +0.000, E1  +414.924, E3 -274308.486}
SPL {X  -159.990, Y  +553.734, Z    +0.000, E1  +414.938, E3 -274319.573}
SPL {X  -159.990, Y  +564.956, Z    +0.000, E1  +414.973, E3 -274336.244}
SPL {X  -159.990, Y  +577.902, Z    +0.000, E1  +414.969, E3 -274355.534}
SPL {X  -159.990, Y  +588.063, Z    +0.000, E1  +414.931, E3 -274370.725}
SPL {X  -159.990, Y  +595.273, Z    +0.000, E1  +414.928, E3 -274381.448}
SPL {X  -159.990, Y  +602.326, Z    +0.000, E1  +414.932, E3 -274391.949}
SPL {X  -159.990, Y  +609.708, Z    +0.000, E1  +414.930, E3 -274402.955}
SPL {X  -159.990, Y  +618.088, Z    +0.000, E1  +414.948, E3 -274415.384}
SPL {X  -159.990, Y  +625.928, Z    +0.000, E1  +414.931, E3 -274427.080}
SPL {X  -159.990, Y  +635.803, Z    +0.000, E1  +414.980, E3 -274441.708}
SPL {X  -159.990, Y  +646.303, Z    +0.000, E1  +414.946, E3 -274457.379}
SPL {X  -159.990, Y  +656.335, Z    +0.000, E1  +414.969, E3 -274472.281}
SPL {X  -159.990, Y  +664.577, Z    +0.000, E1  +414.924, E3 -274484.658}
SPL {X  -159.989, Y  +672.128, Z    +0.000, E1  +414.946, E3 -274495.875}
SPL {X  -159.636, Y  +682.136, Z    +0.000, E1  +414.901, E3 -274511.133}
SPL {X  -158.805, Y  +690.934, Z    +0.000, E1  +414.742, E3 -274525.144}
SPL {X  -157.890, Y  +697.337, Z    +0.000, E1  +414.571, E3 -274535.665}
SPL {X  -156.492, Y  +704.774, Z    +0.000, E1  +414.365, E3 -274548.144}
SPL {X  -154.917, Y  +711.470, Z    +0.000, E1  +414.052, E3 -274559.804}
SPL {X  -153.204, Y  +717.603, Z    +0.000, E1  +413.775, E3 -274570.650}
SPL {X  -151.355, Y  +723.351, Z    +0.000, E1  +413.415, E3 -274581.121}
SPL {X  -148.967, Y  +729.859, Z    +0.000, E1  +413.026, E3 -274593.133}
SPL {X  -145.862, Y  +737.236, Z    +0.000, E1  +412.427, E3 -274607.188}
SPL {X  -142.777, Y  +743.691, Z    +0.000, E1  +411.831, E3 -274619.731}
SPL {X  -132.301, Y  +761.463, Z    +0.000, E1  +405.510, E3 -274699.016}
ENDSPLINE

SPLINE
SPL {X  -145.877, Y  +737.201, Z    +0.000, E1  +394.468, E3 -274782.127}
SPL {X  -152.550, Y  +719.721, Z    +0.000, E1  +387.728, E3 -274797.616}
SPL {X  -157.145, Y  +701.536, Z    +0.000, E1  +379.368, E3 -274807.071}
SPL {X  -159.035, Y  +688.952, Z    +0.000, E1  +372.676, E3 -274811.112}
SPL {X  -159.756, Y  +680.154, Z    +0.000, E1  +367.520, E3 -274812.838}
SPL {X  -159.986, Y  +672.560, Z    +0.000, E1  +362.636, E3 -274813.736}
SPL {X  -159.990, Y  +669.364, Z    +0.000, E1  +360.170, E3 -274813.944}
SPL {X  -159.990, Y  +667.647, Z    +0.000, E1  +358.660, E3 -274814.042}
SPL {X  -159.990, Y  +664.070, Z    +0.000, E1  +354.975, E3 -274814.331}
SPL {X  -159.990, Y  +656.953, Z    +0.000, E1  +346.040, E3 -274815.397}
SPL {X  -159.990, Y  +644.589, Z    +0.000, E1  +330.989, E3 -274818.809}
SPL {X  -159.990, Y  +605.095, Z    +0.000, E1  +310.486, E3 -274843.900}
SPL {X  -159.990, Y  +546.155, Z    +0.000, E1  +305.539, E3 -274906.658}
SPL {X  -159.990, Y  +539.348, Z    +0.000, E1  +305.531, E3 -274916.962}
SPL {X  -159.990, Y  +530.752, Z    +0.000, E1  +305.518, E3 -274929.969}
SPL {X  -159.990, Y  +522.797, Z    +0.000, E1  +305.537, E3 -274942.052}
SPL {X  -159.990, Y  +515.332, Z    +0.000, E1  +305.526, E3 -274953.341}
SPL {X  -159.990, Y  +508.047, Z    +0.000, E1  +305.531, E3 -274964.358}
SPL {X  -159.990, Y  +499.403, Z    +0.000, E1  +305.488, E3 -274977.397}
SPL {X  -159.990, Y  +479.413, Z    +0.000, E1  +302.719, E3 -274988.542}
SPL {X  -159.990, Y  +454.926, Z    +0.000, E1  +299.433, E3 -274997.649}
SPL {X  -159.990, Y  +449.697, Z    +0.000, E1  +300.191, E3 -275009.112}
SPL {X  -159.990, Y  +445.847, Z    +0.000, E1  +300.905, E3 -275018.734}
SPL {X  -159.990, Y  +439.266, Z    +0.000, E1  +301.568, E3 -275031.818}
SPL {X  -159.990, Y  +432.883, Z    +0.000, E1  +302.386, E3 -275045.508}
SPL {X  -159.990, Y  +429.044, Z    +0.000, E1  +303.109, E3 -275055.398}
SPL {X  -159.990, Y  +425.222, Z    +0.000, E1  +304.101, E3 -275067.295}
SPL {X  -159.990, Y  +420.083, Z    +0.000, E1  +304.918, E3 -275079.871}
SPL {X  -159.990, Y  +412.567, Z    +0.000, E1  +305.072, E3 -275092.095}
SPL {X  -159.990, Y  +402.790, Z    +0.000, E1  +305.070, E3 -275106.689}
SPL {X  -159.990, Y  +391.119, Z    +0.000, E1  +305.052, E3 -275124.067}
SPL {X  -159.988, Y  +381.720, Z    +0.000, E1  +305.103, E3 -275138.174}
SPL {X  -159.786, Y  +374.425, Z    +0.000, E1  +305.121, E3 -275149.222}
SPL {X  -159.015, Y  +364.863, Z    +0.000, E1  +305.220, E3 -275164.239}
SPL {X  -157.966, Y  +357.131, Z    +0.000, E1  +305.441, E3 -275176.929}
SPL {X  -156.775, Y  +350.586, Z    +0.000, E1  +305.627, E3 -275187.903}
SPL {X  -155.027, Y  +342.959, Z    +0.000, E1  +305.926, E3 -275201.076}
SPL {X  -152.882, Y  +335.340, Z    +0.000, E1  +306.305, E3 -275214.618}
SPL {X  -150.681, Y  +328.723, Z    +0.000, E1  +306.710, E3 -275226.713}
SPL {X  -148.661, Y  +323.366, Z    +0.000, E1  +307.100, E3 -275236.722}
SPL {X  -147.089, Y  +319.560, Z    +0.000, E1  +307.396, E3 -275243.937}
SPL {X  -145.161, Y  +315.232, Z    +0.000, E1  +307.745, E3 -275252.217}
SPL {X  -142.534, Y  +309.830, Z    +0.000, E1  +308.237, E3 -275262.723}
SPL {X  -132.342, Y  +292.599, Z    +0.000, E1  +315.826, E3 -275360.011}
ENDSPLINE

SPLINE
SPL {X  -151.238, Y  +330.309, Z    +0.000, E1  +330.693, E3 -275433.167}
SPL {X  -156.949, Y  +351.453, Z    +0.000, E1  +340.161, E3 -275445.328}
SPL {X  -159.024, Y  +364.945, Z    +0.000, E1  +347.297, E3 -275449.746}
SPL {X  -159.878, Y  +376.512, Z    +0.000, E1  +354.071, E3 -275451.998}
SPL {X  -159.990, Y  +383.659, Z    +0.000, E1  +358.950, E3 -275452.692}
SPL {X  -159.990, Y  +387.327, Z    +0.000, E1  +362.137, E3 -275452.925}
SPL {X  -159.990, Y  +390.622, Z    +0.000, E1  +365.876, E3 -275453.218}
SPL {X  -159.990, Y  +394.493, Z    +0.000, E1  +370.512, E3 -275453.741}
SPL {X  -159.990, Y  +401.377, Z    +0.000, E1  +379.398, E3 -275455.196}
SPL {X  -159.990, Y  +411.365, Z    +0.000, E1  +390.630, E3 -275458.404}
SPL {X  -159.990, Y  +450.467, Z    +0.000, E1  +410.183, E3 -275482.053}
SPL {X  -159.990, Y  +509.934, Z    +0.000, E1  +414.923, E3 -275544.672}
SPL {X  -159.990, Y  +516.848, Z    +0.000, E1  +414.930, E3 -275554.960}
SPL {X  -159.990, Y  +524.818, Z    +0.000, E1  +414.933, E3 -275566.832}
SPL {X  -159.990, Y  +532.100, Z    +0.000, E1  +414.924, E3 -275577.685}
SPL {X  -159.990, Y  +539.391, Z    +0.000, E1  +414.933, E3 -275588.537}
SPL {X  -159.990, Y  +546.283, Z    +0.000, E1  +414.924, E3 -275598.809}
SPL {X  -159.990, Y  +553.734, Z    +0.000, E1  +414.938, E3 -275609.895}
SPL {X  -159.990, Y  +564.956, Z    +0.000, E1  +414.973, E3 -275626.567}
SPL {X  -159.990, Y  +577.902, Z    +0.000, E1  +414.969, E3 -275645.856}
SPL {X  -159.990, Y  +588.063, Z    +0.000, E1  +414.931, E3 -275661.047}
SPL {X  -159.990, Y  +595.273, Z    +0.000, E1  +414.928, E3 -275671.771}
SPL {X  -159.990, Y  +602.326, Z    +0.000, E1  +414.932, E3 -275682.271}
SPL {X  -159.990, Y  +609.708, Z    +0.000, E1  +414.930, E3 -275693.278}
SPL {X  -159.990, Y  +618.088, Z    +0.000, E1  +414.948, E3 -275705.707}
SPL {X  -159.990, Y  +625.928, Z    +0.000, E1  +414.931, E3 -275717.403}
SPL {X  -159.990, Y  +635.803, Z    +0.000, E1  +414.980, E3 -275732.031}
SPL {X  -159.990, Y  +646.303, Z    +0.000, E1  +414.946, E3 -275747.701}
SPL {X  -159.990, Y  +653.312, Z    +0.000, E1  +414.932, E3 -275758.153}
SPL {X  -159.990, Y  +658.943, Z    +0.000, E1  +414.931, E3 -275766.551}
SPL {X  -159.990, Y  +667.151, Z    +0.000, E1  +414.954, E3 -275778.770}
SPL {X  -159.885, Y  +677.285, Z    +0.000, E1  +414.936, E3 -275793.965}
SPL {X  -159.482, Y  +684.244, Z    +0.000, E1  +414.840, E3 -275804.817}
SPL {X  -158.805, Y  +690.934, Z    +0.000, E1  +414.742, E3 -275815.466}
SPL {X  -157.890, Y  +697.337, Z    +0.000, E1  +414.571, E3 -275825.988}
SPL {X  -156.492, Y  +704.774, Z    +0.000, E1  +414.365, E3 -275838.467}
SPL {X  -154.917, Y  +711.470, Z    +0.000, E1  +414.052, E3 -275850.127}
SPL {X  -153.561, Y  +716.398, Z    +0.000, E1  +413.816, E3 -275858.848}
SPL {X  -151.715, Y  +722.287, Z    +0.000, E1  +413.503, E3 -275869.464}
SPL {X  -148.967, Y  +729.859, Z    +0.000, E1  +413.026, E3 -275883.456}
SPL {X  -145.862, Y  +737.236, Z    +0.000, E1  +412.427, E3 -275897.510}
SPL {X  -142.777, Y  +743.691, Z    +0.000, E1  +411.831, E3 -275910.054}
SPL {X  -132.301, Y  +761.463, Z    +0.000, E1  +405.510, E3 -275989.338}
ENDSPLINE

SPLINE
SPL {X  -145.877, Y  +737.201, Z    +0.000, E1  +394.468, E3 -276072.449}
SPL {X  -152.550, Y  +719.721, Z    +0.000, E1  +387.728, E3 -276087.939}
SPL {X  -157.145, Y  +701.536, Z    +0.000, E1  +379.368, E3 -276097.393}
SPL {X  -159.035, Y  +688.952, Z    +0.000, E1  +372.676, E3 -276101.434}
SPL {X  -159.756, Y  +680.154, Z    +0.000, E1  +367.520, E3 -276103.161}
SPL {X  -159.986, Y  +672.560, Z    +0.000, E1  +362.636, E3 -276104.059}
SPL {X  -159.990, Y  +668.344, Z    +0.000, E1  +359.382, E3 -276104.325}
SPL {X  -159.990, Y  +664.070, Z    +0.000, E1  +354.975, E3 -276104.653}
SPL {X  -159.990, Y  +656.953, Z    +0.000, E1  +346.040, E3 -276105.720}
SPL {X  -159.990, Y  +644.589, Z    +0.000, E1  +330.989, E3 -276109.131}
SPL {X  -159.990, Y  +605.095, Z    +0.000, E1  +310.486, E3 -276134.222}
SPL {X  -159.990, Y  +546.155, Z    +0.000, E1  +305.539, E3 -276196.981}
SPL {X  -159.990, Y  +539.348, Z    +0.000, E1  +305.531, E3 -276207.285}
SPL {X  -159.990, Y  +530.752, Z    +0.000, E1  +305.518, E3 -276220.292}
SPL {X  -159.990, Y  +522.797, Z    +0.000, E1  +305.537, E3 -276232.375}
SPL {X  -159.990, Y  +515.332, Z    +0.000, E1  +305.526, E3 -276243.664}
SPL {X  -159.990, Y  +508.047, Z    +0.000, E1  +305.531, E3 -276254.681}
SPL {X  -159.990, Y  +501.296, Z    +0.000, E1  +305.518, E3 -276264.902}
SPL {X  -159.990, Y  +487.558, Z    +0.000, E1  +304.151, E3 -276276.532}
SPL {X  -159.990, Y  +454.926, Z    +0.000, E1  +299.433, E3 -276287.972}
SPL {X  -159.990, Y  +449.697, Z    +0.000, E1  +300.191, E3 -276299.434}
SPL {X  -159.990, Y  +445.847, Z    +0.000, E1  +300.905, E3 -276309.057}
SPL {X  -159.990, Y  +439.266, Z    +0.000, E1  +301.568, E3 -276322.140}
SPL {X  -159.990, Y  +432.883, Z    +0.000, E1  +302.386, E3 -276335.831}
SPL {X  -159.990, Y  +429.044, Z    +0.000, E1  +303.109, E3 -276345.721}
SPL {X  -159.990, Y  +425.222, Z    +0.000, E1  +304.101, E3 -276357.618}
SPL {X  -159.990, Y  +418.562, Z    +0.000, E1  +304.950, E3 -276372.776}
SPL {X  -159.990, Y  +407.911, Z    +0.000, E1  +305.062, E3 -276389.367}
SPL {X  -159.990, Y  +400.284, Z    +0.000, E1  +305.103, E3 -276400.801}
SPL {X  -159.990, Y  +391.119, Z    +0.000, E1  +305.052, E3 -276414.389}
SPL {X  -159.988, Y  +381.720, Z    +0.000, E1  +305.103, E3 -276428.497}
SPL {X  -159.786, Y  +374.425, Z    +0.000, E1  +305.121, E3 -276439.545}
SPL {X  -159.015, Y  +364.863, Z    +0.000, E1  +305.220, E3 -276454.561}
SPL {X  -157.966, Y  +357.131, Z    +0.000, E1  +305.441, E3 -276467.251}
SPL {X  -156.775, Y  +350.586, Z    +0.000, E1  +305.627, E3 -276478.225}
SPL {X  -155.027, Y  +342.959, Z    +0.000, E1  +305.926, E3 -276491.398}
SPL {X  -152.882, Y  +335.340, Z    +0.000, E1  +306.305, E3 -276504.941}
SPL {X  -150.681, Y  +328.723, Z    +0.000, E1  +306.710, E3 -276517.035}
SPL {X  -148.661, Y  +323.366, Z    +0.000, E1  +307.100, E3 -276527.045}
SPL {X  -147.089, Y  +319.560, Z    +0.000, E1  +307.396, E3 -276534.260}
SPL {X  -145.161, Y  +315.232, Z    +0.000, E1  +307.745, E3 -276542.540}
SPL {X  -142.534, Y  +309.830, Z    +0.000, E1  +308.237, E3 -276553.045}
SPL {X  -132.342, Y  +292.599, Z    +0.000, E1  +315.826, E3 -276650.333}
ENDSPLINE

SPLINE
SPL {X  -151.238, Y  +330.309, Z    +0.000, E1  +330.693, E3 -276723.490}
SPL {X  -156.949, Y  +351.453, Z    +0.000, E1  +340.161, E3 -276735.651}
SPL {X  -159.024, Y  +364.945, Z    +0.000, E1  +347.297, E3 -276740.069}
SPL {X  -159.758, Y  +373.891, Z    +0.000, E1  +352.513, E3 -276741.957}
SPL {X  -159.985, Y  +381.208, Z    +0.000, E1  +357.184, E3 -276742.840}
SPL {X  -159.990, Y  +384.493, Z    +0.000, E1  +359.676, E3 -276743.065}
SPL {X  -159.990, Y  +387.327, Z    +0.000, E1  +362.137, E3 -276743.248}
SPL {X  -159.990, Y  +392.053, Z    +0.000, E1  +367.477, E3 -276743.713}
SPL {X  -159.990, Y  +396.158, Z    +0.000, E1  +372.775, E3 -276744.338}
SPL {X  -159.990, Y  +401.377, Z    +0.000, E1  +379.398, E3 -276745.518}
SPL {X  -159.990, Y  +411.365, Z    +0.000, E1  +390.630, E3 -276748.727}
SPL {X  -159.990, Y  +450.467, Z    +0.000, E1  +410.183, E3 -276772.376}
SPL {X  -159.990, Y  +509.934, Z    +0.000, E1  +414.923, E3 -276834.995}
SPL {X  -159.990, Y  +516.848, Z    +0.000, E1  +414.930, E3 -276845.283}
SPL {X  -159.990, Y  +524.818, Z    +0.000, E1  +414.933, E3 -276857.155}
SPL {X  -159.990, Y  +532.100, Z    +0.000, E1  +414.924, E3 -276868.008}
SPL {X  -159.990, Y  +539.391, Z    +0.000, E1  +414.933, E3 -276878.860}
SPL {X  -159.990, Y  +546.283, Z    +0.000, E1  +414.924, E3 -276889.131}
SPL {X  -159.990, Y  +553.734, Z    +0.000, E1  +414.938, E3 -276900.218}
SPL {X  -159.990, Y  +564.956, Z    +0.000, E1  +414.973, E3 -276916.889}
SPL {X  -159.990, Y  +577.902, Z    +0.000, E1  +414.969, E3 -276936.179}
SPL {X  -159.990, Y  +588.063, Z    +0.000, E1  +414.931, E3 -276951.370}
SPL {X  -159.990, Y  +595.273, Z    +0.000, E1  +414.928, E3 -276962.093}
SPL {X  -159.990, Y  +602.326, Z    +0.000, E1  +414.932, E3 -276972.594}
SPL {X  -159.990, Y  +609.708, Z    +0.000, E1  +414.930, E3 -276983.600}
SPL {X  -159.990, Y  +618.088, Z    +0.000, E1  +414.948, E3 -276996.029}
SPL {X  -159.990, Y  +625.928, Z    +0.000, E1  +414.931, E3 -277007.725}
SPL {X  -159.990, Y  +632.991, Z    +0.000, E1  +414.938, E3 -277018.228}
SPL {X  -159.990, Y  +639.033, Z    +0.000, E1  +414.931, E3 -277027.236}
SPL {X  -159.990, Y  +646.303, Z    +0.000, E1  +414.946, E3 -277038.024}
SPL {X  -159.990, Y  +656.335, Z    +0.000, E1  +414.969, E3 -277052.926}
SPL {X  -159.990, Y  +664.577, Z    +0.000, E1  +414.924, E3 -277065.303}
SPL {X  -159.989, Y  +672.128, Z    +0.000, E1  +414.946, E3 -277076.520}
SPL {X  -159.636, Y  +682.136, Z    +0.000, E1  +414.901, E3 -277091.778}
SPL {X  -158.805, Y  +690.934, Z    +0.000, E1  +414.742, E3 -277105.789}
SPL {X  -157.890, Y  +697.337, Z    +0.000, E1  +414.571, E3 -277116.310}
SPL {X  -156.492, Y  +704.774, Z    +0.000, E1  +414.365, E3 -277128.789}
SPL {X  -154.917, Y  +711.470, Z    +0.000, E1  +414.052, E3 -277140.449}
SPL {X  -153.204, Y  +717.603, Z    +0.000, E1  +413.775, E3 -277151.295}
SPL {X  -151.355, Y  +723.351, Z    +0.000, E1  +413.415, E3 -277161.766}
SPL {X  -148.967, Y  +729.859, Z    +0.000, E1  +413.026, E3 -277173.779}
SPL {X  -145.862, Y  +737.236, Z    +0.000, E1  +412.427, E3 -277187.833}
SPL {X  -142.777, Y  +743.691, Z    +0.000, E1  +411.831, E3 -277200.376}
SPL {X  -132.301, Y  +761.463, Z    +0.000, E1  +405.510, E3 -277279.661}
ENDSPLINE

SPLINE
SPL {X  -145.877, Y  +737.201, Z    +0.000, E1  +394.468, E3 -277362.772}
SPL {X  -152.550, Y  +719.721, Z    +0.000, E1  +387.728, E3 -277378.261}
SPL {X  -157.145, Y  +701.536, Z    +0.000, E1  +379.368, E3 -277387.716}
SPL {X  -159.035, Y  +688.952, Z    +0.000, E1  +372.676, E3 -277391.757}
SPL {X  -159.756, Y  +680.154, Z    +0.000, E1  +367.520, E3 -277393.483}
SPL {X  -159.986, Y  +672.560, Z    +0.000, E1  +362.636, E3 -277394.381}
SPL {X  -159.990, Y  +668.344, Z    +0.000, E1  +359.382, E3 -277394.647}
SPL {X  -159.990, Y  +665.430, Z    +0.000, E1  +356.370, E3 -277394.843}
SPL {X  -159.990, Y  +661.750, Z    +0.000, E1  +352.120, E3 -277395.234}
SPL {X  -159.990, Y  +657.656, Z    +0.000, E1  +346.724, E3 -277395.878}
SPL {X  -159.990, Y  +652.023, Z    +0.000, E1  +339.551, E3 -277397.166}
SPL {X  -159.990, Y  +641.935, Z    +0.000, E1  +328.152, E3 -277400.338}
SPL {X  -159.990, Y  +605.095, Z    +0.000, E1  +310.486, E3 -277424.545}
SPL {X  -159.990, Y  +546.155, Z    +0.000, E1  +305.539, E3 -277487.303}
SPL {X  -159.990, Y  +539.348, Z    +0.000, E1  +305.531, E3 -277497.607}
SPL {X  -159.990, Y  +530.752, Z    +0.000, E1  +305.518, E3 -277510.614}
SPL {X  -159.990, Y  +522.797, Z    +0.000, E1  +305.537, E3 -277522.698}
SPL {X  -159.990, Y  +515.332, Z    +0.000, E1  +305.526, E3 -277533.986}
SPL {X  -159.990, Y  +508.047, Z    +0.000, E1  +305.531, E3 -277545.003}
SPL {X  -159.990, Y  +499.403, Z    +0.000, E1  +305.488, E3 -277558.042}
SPL {X  -159.990, Y  +479.413, Z    +0.000, E1  +302.719, E3 -277569.188}
SPL {X  -159.990, Y  +454.926, Z    +0.000, E1  +299.433, E3 -277578.294}
SPL {X  -159.990, Y  +449.697, Z    +0.000, E1  +300.191, E3 -277589.757}
SPL {X  -159.990, Y  +444.026, Z    +0.000, E1  +301.072, E3 -277603.015}
SPL {X  -159.990, Y  +437.596, Z    +0.000, E1  +301.764, E3 -277615.756}
SPL {X  -159.990, Y  +432.883, Z    +0.000, E1  +302.386, E3 -277626.153}
SPL {X  -159.990, Y  +429.044, Z    +0.000, E1  +303.109, E3 -277636.043}
SPL {X  -159.990, Y  +425.222, Z    +0.000, E1  +304.101, E3 -277647.941}
SPL {X  -159.990, Y  +418.562, Z    +0.000, E1  +304.950, E3 -277663.098}
SPL {X  -159.990, Y  +410.722, Z    +0.000, E1  +305.100, E3 -277675.559}
SPL {X  -159.990, Y  +402.790, Z    +0.000, E1  +305.070, E3 -277687.334}
SPL {X  -159.990, Y  +391.119, Z    +0.000, E1  +305.052, E3 -277704.712}
SPL {X  -159.988, Y  +381.720, Z    +0.000, E1  +305.103, E3 -277718.819}
SPL {X  -159.786, Y  +374.425, Z    +0.000, E1  +305.121, E3 -277729.867}
SPL {X  -159.015, Y  +364.863, Z    +0.000, E1  +305.220, E3 -277744.884}
SPL {X  -157.966, Y  +357.131, Z    +0.000, E1  +305.441, E3 -277757.574}
SPL {X  -156.775, Y  +350.586, Z    +0.000, E1  +305.627, E3 -277768.548}
SPL {X  -155.397, Y  +344.442, Z    +0.000, E1  +305.886, E3 -277779.164}
SPL {X  -153.976, Y  +339.046, Z    +0.000, E1  +306.128, E3 -277788.656}
SPL {X  -152.417, Y  +333.859, Z    +0.000, E1  +306.416, E3 -277797.982}
SPL {X  -150.681, Y  +328.723, Z    +0.000, E1  +306.710, E3 -277807.358}
SPL {X  -148.661, Y  +323.366, Z    +0.000, E1  +307.100, E3 -277817.367}
SPL {X  -147.089, Y  +319.560, Z    +0.000, E1  +307.396, E3 -277824.582}
SPL {X  -145.161, Y  +315.232, Z    +0.000, E1  +307.745, E3 -277832.863}
SPL {X  -142.534, Y  +309.830, Z    +0.000, E1  +308.237, E3 -277843.368}
SPL {X  -132.342, Y  +292.599, Z    +0.000, E1  +315.826, E3 -277940.656}
ENDSPLINE

SPLINE
SPL {X  -151.238, Y  +330.309, Z    +0.000, E1  +330.693, E3 -278013.813}
SPL {X  -156.949, Y  +351.453, Z    +0.000, E1  +340.161, E3 -278025.973}
SPL {X  -159.024, Y  +364.945, Z    +0.000, E1  +347.297, E3 -278030.391}
SPL {X  -159.758, Y  +373.891, Z    +0.000, E1  +352.513, E3 -278032.280}
SPL {X  -159.985, Y  +381.208, Z    +0.000, E1  +357.184, E3 -278033.163}
SPL {X  -159.990, Y  +385.261, Z    +0.000, E1  +360.259, E3 -278033.433}
SPL {X  -159.990, Y  +388.094, Z    +0.000, E1  +363.012, E3 -278033.625}
SPL {X  -159.990, Y  +390.622, Z    +0.000, E1  +365.876, E3 -278033.864}
SPL {X  -159.990, Y  +394.493, Z    +0.000, E1  +370.512, E3 -278034.386}
SPL {X  -159.990, Y  +401.377, Z    +0.000, E1  +379.398, E3 -278035.841}
SPL {X  -159.990, Y  +411.365, Z    +0.000, E1  +390.630, E3 -278039.049}
SPL {X  -159.990, Y  +450.467, Z    +0.000, E1  +410.183, E3 -278062.698}
SPL {X  -159.990, Y  +509.934, Z    +0.000, E1  +414.923, E3 -278125.317}
SPL {X  -159.990, Y  +516.848, Z    +0.000, E1  +414.930, E3 -278135.605}
SPL {X  -159.990, Y  +524.818, Z    +0.000, E1  +414.933, E3 -278147.477}
SPL {X  -159.990, Y  +532.100, Z    +0.000, E1  +414.924, E3 -278158.330}
SPL {X  -159.990, Y  +539.391, Z    +0.000, E1  +414.933, E3 -278169.182}
SPL {X  -159.990, Y  +546.283, Z    +0.000, E1  +414.924, E3 -278179.454}
SPL {X  -159.990, Y  +553.734, Z    +0.000, E1  +414.938, E3 -278190.541}
SPL {X  -159.990, Y  +564.956, Z    +0.000, E1  +414.973, E3 -278207.212}
SPL {X  -159.990, Y  +577.902, Z    +0.000, E1  +414.969, E3 -278226.502}
SPL {X  -159.990, Y  +588.063, Z    +0.000, E1  +414.931, E3 -278241.692}
SPL {X  -159.990, Y  +595.273, Z    +0.000, E1  +414.928, E3 -278252.416}
SPL {X  -159.990, Y  +602.326, Z    +0.000, E1  +414.932, E3 -278262.916}
SPL {X  -159.990, Y  +609.708, Z    +0.000, E1  +414.930, E3 -278273.923}
SPL {X  -159.990, Y  +618.088, Z    +0.000, E1  +414.948, E3 -278286.352}
SPL {X  -159.990, Y  +625.928, Z    +0.000, E1  +414.931, E3 -278298.048}
SPL {X  -159.990, Y  +632.991, Z    +0.000, E1  +414.938, E3 -278308.551}
SPL {X  -159.990, Y  +639.033, Z    +0.000, E1  +414.931, E3 -278317.558}
SPL {X  -159.990, Y  +646.303, Z    +0.000, E1  +414.946, E3 -278328.346}
SPL {X  -159.990, Y  +656.335, Z    +0.000, E1  +414.969, E3 -278343.249}
SPL {X  -159.990, Y  +664.577, Z    +0.000, E1  +414.924, E3 -278355.626}
SPL {X  -159.989, Y  +672.128, Z    +0.000, E1  +414.946, E3 -278366.843}
SPL {X  -159.792, Y  +679.466, Z    +0.000, E1  +414.893, E3 -278378.000}
SPL {X  -159.330, Y  +686.016, Z    +0.000, E1  +414.837, E3 -278388.232}
SPL {X  -158.190, Y  +695.432, Z    +0.000, E1  +414.658, E3 -278403.428}
SPL {X  -157.027, Y  +702.151, Z    +0.000, E1  +414.415, E3 -278414.710}
SPL {X  -156.112, Y  +706.513, Z    +0.000, E1  +414.265, E3 -278422.144}
SPL {X  -154.917, Y  +711.470, Z    +0.000, E1  +414.052, E3 -278430.772}
SPL {X  -153.561, Y  +716.398, Z    +0.000, E1  +413.816, E3 -278439.493}
SPL {X  -151.715, Y  +722.287, Z    +0.000, E1  +413.503, E3 -278450.109}
SPL {X  -148.967, Y  +729.859, Z    +0.000, E1  +413.026, E3 -278464.101}
SPL {X  -145.862, Y  +737.236, Z    +0.000, E1  +412.427, E3 -278478.155}
SPL {X  -142.777, Y  +743.691, Z    +0.000, E1  +411.831, E3 -278490.699}
SPL {X  -132.301, Y  +761.463, Z    +0.000, E1  +405.510, E3 -278569.984}
ENDSPLINE

SPLINE
SPL {X  -145.877, Y  +737.201, Z    +0.000, E1  +394.468, E3 -278653.095}
SPL {X  -152.550, Y  +719.721, Z    +0.000, E1  +387.728, E3 -278668.584}
SPL {X  -157.145, Y  +701.536, Z    +0.000, E1  +379.368, E3 -278678.038}
SPL {X  -159.035, Y  +688.952, Z    +0.000, E1  +372.676, E3 -278682.079}
SPL {X  -159.756, Y  +680.154, Z    +0.000, E1  +367.520, E3 -278683.806}
SPL {X  -159.986, Y  +672.560, Z    +0.000, E1  +362.636, E3 -278684.704}
SPL {X  -159.990, Y  +668.344, Z    +0.000, E1  +359.382, E3 -278684.970}
SPL {X  -159.990, Y  +664.070, Z    +0.000, E1  +354.975, E3 -278685.298}
SPL {X  -159.990, Y  +656.953, Z    +0.000, E1  +346.040, E3 -278686.365}
SPL {X  -159.990, Y  +644.589, Z    +0.000, E1  +330.989, E3 -278689.776}
SPL {X  -159.990, Y  +605.095, Z    +0.000, E1  +310.486, E3 -278714.867}
SPL {X  -159.990, Y  +546.155, Z    +0.000, E1  +305.539, E3 -278777.626}
SPL {X  -159.990, Y  +539.348, Z    +0.000, E1  +305.531, E3 -278787.930}
SPL {X  -159.990, Y  +530.752, Z    +0.000, E1  +305.518, E3 -278800.937}
SPL {X  -159.990, Y  +522.797, Z    +0.000, E1  +305.537, E3 -278813.020}
SPL {X  -159.990, Y  +515.332, Z    +0.000, E1  +305.526, E3 -278824.309}
SPL {X  -159.990, Y  +508.047, Z    +0.000, E1  +305.531, E3 -278835.326}
SPL {X  -159.990, Y  +499.403, Z    +0.000, E1  +305.488, E3 -278848.365}
SPL {X  -159.990, Y  +479.413, Z    +0.000, E1  +302.719, E3 -278859.510}
SPL {X  -159.990, Y  +454.926, Z    +0.000, E1  +299.433, E3 -278868.617}
SPL {X  -159.990, Y  +449.697, Z    +0.000, E1  +300.191, E3 -278880.079}
SPL {X  -159.990, Y  +445.847, Z    +0.000, E1  +300.905, E3 -278889.702}
SPL {X  -159.990, Y  +439.266, Z    +0.000, E1  +301.568, E3 -278902.786}
SPL {X  -159.990, Y  +432.883, Z    +0.000, E1  +302.386, E3 -278916.476}
SPL {X  -159.990, Y  +429.044, Z    +0.000, E1  +303.109, E3 -278926.366}
SPL {X  -159.990, Y  +425.222, Z    +0.000, E1  +304.101, E3 -278938.263}
SPL {X  -159.990, Y  +420.083, Z    +0.000, E1  +304.918, E3 -278950.839}
SPL {X  -159.990, Y  +412.567, Z    +0.000, E1  +305.072, E3 -278963.063}
SPL {X  -159.990, Y  +402.790, Z    +0.000, E1  +305.070, E3 -278977.657}
SPL {X  -159.990, Y  +391.119, Z    +0.000, E1  +305.052, E3 -278995.035}
SPL {X  -159.988, Y  +381.720, Z    +0.000, E1  +305.103, E3 -279009.142}
SPL {X  -159.786, Y  +374.425, Z    +0.000, E1  +305.121, E3 -279020.190}
SPL {X  -159.015, Y  +364.863, Z    +0.000, E1  +305.220, E3 -279035.206}
SPL {X  -157.966, Y  +357.131, Z    +0.000, E1  +305.441, E3 -279047.897}
SPL {X  -156.775, Y  +350.586, Z    +0.000, E1  +305.627, E3 -279058.871}
SPL {X  -155.027, Y  +342.959, Z    +0.000, E1  +305.926, E3 -279072.044}
SPL {X  -152.882, Y  +335.340, Z    +0.000, E1  +306.305, E3 -279085.586}
SPL {X  -150.681, Y  +328.723, Z    +0.000, E1  +306.710, E3 -279097.681}
SPL {X  -148.661, Y  +323.366, Z    +0.000, E1  +307.100, E3 -279107.690}
SPL {X  -147.089, Y  +319.560, Z    +0.000, E1  +307.396, E3 -279114.905}
SPL {X  -145.161, Y  +315.232, Z    +0.000, E1  +307.745, E3 -279123.185}
SPL {X  -142.534, Y  +309.830, Z    +0.000, E1  +308.237, E3 -279133.690}
SPL {X  -132.342, Y  +292.599, Z    +0.000, E1  +315.826, E3 -279230.978}
ENDSPLINE

SPLINE
SPL {X  -151.238, Y  +330.309, Z    +0.000, E1  +330.693, E3 -279304.135}
SPL {X  -156.949, Y  +351.453, Z    +0.000, E1  +340.161, E3 -279316.296}
SPL {X  -159.024, Y  +364.945, Z    +0.000, E1  +347.297, E3 -279320.714}
SPL {X  -159.878, Y  +376.512, Z    +0.000, E1  +354.071, E3 -279322.965}
SPL {X  -159.990, Y  +383.659, Z    +0.000, E1  +358.950, E3 -279323.660}
SPL {X  -159.990, Y  +387.327, Z    +0.000, E1  +362.137, E3 -279323.893}
SPL {X  -159.990, Y  +390.622, Z    +0.000, E1  +365.876, E3 -279324.186}
SPL {X  -159.990, Y  +394.493, Z    +0.000, E1  +370.512, E3 -279324.709}
SPL {X  -159.990, Y  +401.377, Z    +0.000, E1  +379.398, E3 -279326.164}
SPL {X  -159.990, Y  +411.365, Z    +0.000, E1  +390.630, E3 -279329.372}
SPL {X  -159.990, Y  +450.467, Z    +0.000, E1  +410.183, E3 -279353.021}
SPL {X  -159.990, Y  +509.934, Z    +0.000, E1  +414.923, E3 -279415.640}
SPL {X  -159.990, Y  +516.848, Z    +0.000, E1  +414.930, E3 -279425.928}
SPL {X  -159.990, Y  +524.818, Z    +0.000, E1  +414.933, E3 -279437.800}
SPL {X  -159.990, Y  +532.100, Z    +0.000, E1  +414.924, E3 -279448.653}
SPL {X  -159.990, Y  +539.391, Z    +0.000, E1  +414.933, E3 -279459.505}
SPL {X  -159.990, Y  +546.283, Z    +0.000, E1  +414.924, E3 -279469.776}
SPL {X  -159.990, Y  +553.734, Z    +0.000, E1  +414.938, E3 -279480.863}
SPL {X  -159.990, Y  +564.956, Z    +0.000, E1  +414.973, E3 -279497.534}
SPL {X  -159.990, Y  +577.902, Z    +0.000, E1  +414.969, E3 -279516.824}
SPL {X  -159.990, Y  +588.063, Z    +0.000, E1  +414.931, E3 -279532.015}
SPL {X  -159.990, Y  +595.273, Z    +0.000, E1  +414.928, E3 -279542.739}
SPL {X  -159.990, Y  +602.326, Z    +0.000, E1  +414.932, E3 -279553.239}
SPL {X  -159.990, Y  +609.708, Z    +0.000, E1  +414.930, E3 -279564.246}
SPL {X  -159.990, Y  +618.088, Z    +0.000, E1  +414.948, E3 -279576.675}
SPL {X  -159.990, Y  +625.928, Z    +0.000, E1  +414.931, E3 -279588.370}
SPL {X  -159.990, Y  +635.803, Z    +0.000, E1  +414.980, E3 -279602.998}
SPL {X  -159.990, Y  +646.303, Z    +0.000, E1  +414.946, E3 -279618.669}
SPL {X  -159.990, Y  +653.312, Z    +0.000, E1  +414.932, E3 -279629.121}
SPL {X  -159.990, Y  +658.943, Z    +0.000, E1  +414.931, E3 -279637.519}
SPL {X  -159.990, Y  +667.151, Z    +0.000, E1  +414.954, E3 -279649.737}
SPL {X  -159.885, Y  +677.285, Z    +0.000, E1  +414.936, E3 -279664.933}
SPL {X  -159.482, Y  +684.244, Z    +0.000, E1  +414.840, E3 -279675.785}
SPL {X  -158.805, Y  +690.934, Z    +0.000, E1  +414.742, E3 -279686.434}
SPL {X  -157.890, Y  +697.337, Z    +0.000, E1  +414.571, E3 -279696.955}
SPL {X  -156.492, Y  +704.774, Z    +0.000, E1  +414.365, E3 -279709.434}
SPL {X  -154.917, Y  +711.470, Z    +0.000, E1  +414.052, E3 -279721.094}
SPL {X  -153.561, Y  +716.398, Z    +0.000, E1  +413.816, E3 -279729.816}
SPL {X  -151.715, Y  +722.287, Z    +0.000, E1  +413.503, E3 -279740.432}
SPL {X  -148.967, Y  +729.859, Z    +0.000, E1  +413.026, E3 -279754.424}
SPL {X  -145.862, Y  +737.236, Z    +0.000, E1  +412.427, E3 -279768.478}
SPL {X  -142.777, Y  +743.691, Z    +0.000, E1  +411.831, E3 -279781.021}
SPL {X  -132.301, Y  +761.463, Z    +0.000, E1  +405.510, E3 -279860.306}
ENDSPLINE

SPLINE
SPL {X  -145.877, Y  +737.201, Z    +0.000, E1  +394.468, E3 -279943.417}
SPL {X  -152.550, Y  +719.721, Z    +0.000, E1  +387.728, E3 -279958.906}
SPL {X  -157.145, Y  +701.536, Z    +0.000, E1  +379.368, E3 -279968.361}
SPL {X  -159.035, Y  +688.952, Z    +0.000, E1  +372.676, E3 -279972.402}
SPL {X  -159.756, Y  +680.154, Z    +0.000, E1  +367.520, E3 -279974.128}
SPL {X  -159.986, Y  +672.560, Z    +0.000, E1  +362.636, E3 -279975.026}
SPL {X  -159.990, Y  +668.344, Z    +0.000, E1  +359.382, E3 -279975.293}
SPL {X  -159.990, Y  +664.070, Z    +0.000, E1  +354.975, E3 -279975.621}
SPL {X  -159.990, Y  +656.953, Z    +0.000, E1  +346.040, E3 -279976.687}
SPL {X  -159.990, Y  +644.589, Z    +0.000, E1  +330.989, E3 -279980.099}
SPL {X  -159.990, Y  +605.095, Z    +0.000, E1  +310.486, E3 -280005.190}
SPL {X  -159.990, Y  +546.155, Z    +0.000, E1  +305.539, E3 -280067.948}
SPL {X  -159.990, Y  +539.348, Z    +0.000, E1  +305.531, E3 -280078.252}
SPL {X  -159.990, Y  +530.752, Z    +0.000, E1  +305.518, E3 -280091.260}
SPL {X  -159.990, Y  +522.797, Z    +0.000, E1  +305.537, E3 -280103.343}
SPL {X  -159.990, Y  +515.332, Z    +0.000, E1  +305.526, E3 -280114.632}
SPL {X  -159.990, Y  +508.047, Z    +0.000, E1  +305.531, E3 -280125.648}
SPL {X  -159.990, Y  +501.296, Z    +0.000, E1  +305.518, E3 -280135.870}
SPL {X  -159.990, Y  +487.558, Z    +0.000, E1  +304.151, E3 -280147.500}
SPL {X  -159.990, Y  +454.926, Z    +0.000, E1  +299.433, E3 -280158.939}
SPL {X  -159.990, Y  +449.697, Z    +0.000, E1  +300.191, E3 -280170.402}
SPL {X  -159.990, Y  +445.847, Z    +0.000, E1  +300.905, E3 -280180.025}
SPL {X  -159.990, Y  +439.266, Z    +0.000, E1  +301.568, E3 -280193.108}
SPL {X  -159.990, Y  +432.883, Z    +0.000, E1  +302.386, E3 -280206.798}
SPL {X  -159.990, Y  +429.044, Z    +0.000, E1  +303.109, E3 -280216.689}
SPL {X  -159.990, Y  +425.222, Z    +0.000, E1  +304.101, E3 -280228.586}
SPL {X  -159.990, Y  +418.562, Z    +0.000, E1  +304.950, E3 -280243.743}
SPL {X  -159.990, Y  +407.911, Z    +0.000, E1  +305.062, E3 -280260.335}
SPL {X  -159.990, Y  +400.284, Z    +0.000, E1  +305.103, E3 -280271.769}
SPL {X  -159.990, Y  +391.119, Z    +0.000, E1  +305.052, E3 -280285.357}
SPL {X  -159.988, Y  +381.720, Z    +0.000, E1  +305.103, E3 -280299.464}
SPL {X  -159.786, Y  +374.425, Z    +0.000, E1  +305.121, E3 -280310.513}
SPL {X  -159.015, Y  +364.863, Z    +0.000, E1  +305.220, E3 -280325.529}
SPL {X  -157.966, Y  +357.131, Z    +0.000, E1  +305.441, E3 -280338.219}
SPL {X  -156.775, Y  +350.586, Z    +0.000, E1  +305.627, E3 -280349.193}
SPL {X  -155.027, Y  +342.959, Z    +0.000, E1  +305.926, E3 -280362.366}
SPL {X  -152.882, Y  +335.340, Z    +0.000, E1  +306.305, E3 -280375.909}
SPL {X  -150.681, Y  +328.723, Z    +0.000, E1  +306.710, E3 -280388.003}
SPL {X  -148.661, Y  +323.366, Z    +0.000, E1  +307.100, E3 -280398.012}
SPL {X  -147.089, Y  +319.560, Z    +0.000, E1  +307.396, E3 -280405.227}
SPL {X  -145.161, Y  +315.232, Z    +0.000, E1  +307.745, E3 -280413.508}
SPL {X  -142.534, Y  +309.830, Z    +0.000, E1  +308.237, E3 -280424.013}
SPL {X  -132.342, Y  +292.599, Z    +0.000, E1  +315.826, E3 -280521.301}
ENDSPLINE

SPLINE
SPL {X  -151.238, Y  +330.309, Z    +0.000, E1  +330.693, E3 -280594.458}
SPL {X  -156.949, Y  +351.453, Z    +0.000, E1  +340.161, E3 -280606.619}
SPL {X  -159.024, Y  +364.945, Z    +0.000, E1  +347.297, E3 -280611.036}
SPL {X  -159.758, Y  +373.891, Z    +0.000, E1  +352.513, E3 -280612.925}
SPL {X  -159.985, Y  +381.208, Z    +0.000, E1  +357.184, E3 -280613.808}
SPL {X  -159.990, Y  +384.493, Z    +0.000, E1  +359.676, E3 -280614.033}
SPL {X  -159.990, Y  +387.327, Z    +0.000, E1  +362.137, E3 -280614.215}
SPL {X  -159.990, Y  +392.053, Z    +0.000, E1  +367.477, E3 -280614.680}
SPL {X  -159.990, Y  +396.158, Z    +0.000, E1  +372.775, E3 -280615.306}
SPL {X  -159.990, Y  +401.377, Z    +0.000, E1  +379.398, E3 -280616.486}
SPL {X  -159.990, Y  +411.365, Z    +0.000, E1  +390.630, E3 -280619.695}
SPL {X  -159.990, Y  +450.467, Z    +0.000, E1  +410.183, E3 -280643.343}
SPL {X  -159.990, Y  +509.934, Z    +0.000, E1  +414.923, E3 -280705.962}
SPL {X  -159.990, Y  +516.848, Z    +0.000, E1  +414.930, E3 -280716.250}
SPL {X  -159.990, Y  +524.818, Z    +0.000, E1  +414.933, E3 -280728.122}
SPL {X  -159.990, Y  +532.100, Z    +0.000, E1  +414.924, E3 -280738.975}
SPL {X  -159.990, Y  +539.391, Z    +0.000, E1  +414.933, E3 -280749.827}
SPL {X  -159.990, Y  +546.283, Z    +0.000, E1  +414.924, E3 -280760.099}
SPL {X  -159.990, Y  +553.734, Z    +0.000, E1  +414.938, E3 -280771.186}
SPL {X  -159.990, Y  +564.956, Z    +0.000, E1  +414.973, E3 -280787.857}
SPL {X  -159.990, Y  +577.902, Z    +0.000, E1  +414.969, E3 -280807.147}
SPL {X  -159.990, Y  +588.063, Z    +0.000, E1  +414.931, E3 -280822.338}
SPL {X  -159.990, Y  +595.273, Z    +0.000, E1  +414.928, E3 -280833.061}
SPL {X  -159.990, Y  +602.326, Z    +0.000, E1  +414.932, E3 -280843.562}
SPL {X  -159.990, Y  +609.708, Z    +0.000, E1  +414.930, E3 -280854.568}
SPL {X  -159.990, Y  +618.088, Z    +0.000, E1  +414.948, E3 -280866.997}
SPL {X  -159.990, Y  +625.928, Z    +0.000, E1  +414.931, E3 -280878.693}
SPL {X  -159.990, Y  +632.991, Z    +0.000, E1  +414.938, E3 -280889.196}
SPL {X  -159.990, Y  +639.033, Z    +0.000, E1  +414.931, E3 -280898.204}
SPL {X  -159.990, Y  +646.303, Z    +0.000, E1  +414.946, E3 -280908.992}
SPL {X  -159.990, Y  +656.335, Z    +0.000, E1  +414.969, E3 -280923.894}
SPL {X  -159.990, Y  +664.577, Z    +0.000, E1  +414.924, E3 -280936.271}
SPL {X  -159.989, Y  +672.128, Z    +0.000, E1  +414.946, E3 -280947.488}
SPL {X  -159.636, Y  +682.136, Z    +0.000, E1  +414.901, E3 -280962.746}
SPL {X  -158.805, Y  +690.934, Z    +0.000, E1  +414.742, E3 -280976.757}
SPL {X  -157.890, Y  +697.337, Z    +0.000, E1  +414.571, E3 -280987.278}
SPL {X  -156.492, Y  +704.774, Z    +0.000, E1  +414.365, E3 -280999.757}
SPL {X  -154.917, Y  +711.470, Z    +0.000, E1  +414.052, E3 -281011.417}
SPL {X  -153.204, Y  +717.603, Z    +0.000, E1  +413.775, E3 -281022.263}
SPL {X  -151.355, Y  +723.351, Z    +0.000, E1  +413.415, E3 -281032.734}
SPL {X  -148.967, Y  +729.859, Z    +0.000, E1  +413.026, E3 -281044.746}
SPL {X  -145.862, Y  +737.236, Z    +0.000, E1  +412.427, E3 -281058.801}
SPL {X  -142.777, Y  +743.691, Z    +0.000, E1  +411.831, E3 -281071.344}
SPL {X  -132.301, Y  +761.463, Z    +0.000, E1  +405.510, E3 -281150.629}
ENDSPLINE

SPLINE
SPL {X  -145.877, Y  +737.201, Z    +0.000, E1  +394.468, E3 -281233.740}
SPL {X  -152.550, Y  +719.721, Z    +0.000, E1  +387.728, E3 -281249.229}
SPL {X  -157.145, Y  +701.536, Z    +0.000, E1  +379.368, E3 -281258.684}
SPL {X  -159.035, Y  +688.952, Z    +0.000, E1  +372.676, E3 -281262.725}
SPL {X  -159.756, Y  +680.154, Z    +0.000, E1  +367.520, E3 -281264.451}
SPL {X  -159.986, Y  +672.560, Z    +0.000, E1  +362.636, E3 -281265.349}
SPL {X  -159.990, Y  +668.344, Z    +0.000, E1  +359.382, E3 -281265.615}
SPL {X  -159.990, Y  +664.070, Z    +0.000, E1  +354.975, E3 -281265.944}
SPL {X  -159.990, Y  +656.953, Z    +0.000, E1  +346.040, E3 -281267.010}
SPL {X  -159.990, Y  +644.589, Z    +0.000, E1  +330.989, E3 -281270.422}
SPL {X  -159.990, Y  +605.095, Z    +0.000, E1  +310.486, E3 -281295.512}
SPL {X  -159.990, Y  +546.155, Z    +0.000, E1  +305.539, E3 -281358.271}
SPL {X  -159.990, Y  +539.348, Z    +0.000, E1  +305.531, E3 -281368.575}
SPL {X  -159.990, Y  +530.752, Z    +0.000, E1  +305.518, E3 -281381.582}
SPL {X  -159.990, Y  +522.797, Z    +0.000, E1  +305.537, E3 -281393.665}
SPL {X  -159.990, Y  +515.332, Z    +0.000, E1  +305.526, E3 -281404.954}
SPL {X  -159.990, Y  +508.047, Z    +0.000, E1  +305.531, E3 -281415.971}
SPL {X  -159.990, Y  +501.296, Z    +0.000, E1  +305.518, E3 -281426.192}
SPL {X  -159.990, Y  +487.558, Z    +0.000, E1  +304.151, E3 -281437.823}
SPL {X  -159.990, Y  +454.926, Z    +0.000, E1  +299.433, E3 -281449.262}
SPL {X  -159.990, Y  +449.697, Z    +0.000, E1  +300.191, E3 -281460.724}
SPL {X  -159.990, Y  +445.847, Z    +0.000, E1  +300.905, E3 -281470.347}
SPL {X  -159.990, Y  +439.266, Z    +0.000, E1  +301.568, E3 -281483.431}
SPL {X  -159.990, Y  +432.883, Z    +0.000, E1  +302.386, E3 -281497.121}
SPL {X  -159.990, Y  +428.299, Z    +0.000, E1  +303.316, E3 -281509.525}
SPL {X  -159.990, Y  +424.402, Z    +0.000, E1  +304.297, E3 -281521.200}
SPL {X  -159.990, Y  +418.562, Z    +0.000, E1  +304.950, E3 -281534.066}
SPL {X  -159.990, Y  +410.722, Z    +0.000, E1  +305.100, E3 -281546.527}
SPL {X  -159.990, Y  +402.790, Z    +0.000, E1  +305.070, E3 -281558.302}
SPL {X  -159.990, Y  +391.119, Z    +0.000, E1  +305.052, E3 -281575.680}
SPL {X  -159.988, Y  +381.720, Z    +0.000, E1  +305.103, E3 -281589.787}
SPL {X  -159.786, Y  +374.425, Z    +0.000, E1  +305.121, E3 -281600.835}
SPL {X  -159.184, Y  +366.462, Z    +0.000, E1  +305.220, E3 -281613.336}
SPL {X  -158.166, Y  +358.413, Z    +0.000, E1  +305.386, E3 -281626.391}
SPL {X  -156.775, Y  +350.586, Z    +0.000, E1  +305.627, E3 -281639.516}
SPL {X  -155.027, Y  +342.959, Z    +0.000, E1  +305.926, E3 -281652.689}
SPL {X  -152.882, Y  +335.340, Z    +0.000, E1  +306.305, E3 -281666.231}
SPL {X  -150.681, Y  +328.723, Z    +0.000, E1  +306.710, E3 -281678.326}
SPL {X  -147.884, Y  +321.449, Z    +0.000, E1  +307.200, E3 -281691.899}
SPL {X  -145.161, Y  +315.232, Z    +0.000, E1  +307.745, E3 -281703.830}
SPL {X  -142.534, Y  +309.830, Z    +0.000, E1  +308.237, E3 -281714.335}
SPL {X  -132.342, Y  +292.599, Z    +0.000, E1  +315.826, E3 -281811.624}
ENDSPLINE

SPLINE
SPL {X  -151.238, Y  +330.309, Z    +0.000, E1  +330.693, E3 -281884.780}
SPL {X  -156.949, Y  +351.453, Z    +0.000, E1  +340.161, E3 -281896.941}
SPL {X  -159.024, Y  +364.945, Z    +0.000, E1  +347.297, E3 -281901.359}
SPL {X  -159.878, Y  +376.512, Z    +0.000, E1  +354.071, E3 -281903.610}
SPL {X  -159.990, Y  +383.659, Z    +0.000, E1  +358.950, E3 -281904.305}
SPL {X  -159.990, Y  +387.327, Z    +0.000, E1  +362.137, E3 -281904.538}
SPL {X  -159.990, Y  +390.622, Z    +0.000, E1  +365.876, E3 -281904.831}
SPL {X  -159.990, Y  +394.493, Z    +0.000, E1  +370.512, E3 -281905.354}
SPL {X  -159.990, Y  +401.377, Z    +0.000, E1  +379.398, E3 -281906.809}
SPL {X  -159.990, Y  +411.365, Z    +0.000, E1  +390.630, E3 -281910.017}
SPL {X  -159.990, Y  +450.467, Z    +0.000, E1  +410.183, E3 -281933.666}
SPL {X  -159.990, Y  +509.934, Z    +0.000, E1  +414.923, E3 -281996.285}
SPL {X  -159.990, Y  +516.848, Z    +0.000, E1  +414.930, E3 -282006.573}
SPL {X  -159.990, Y  +524.818, Z    +0.000, E1  +414.933, E3 -282018.445}
SPL {X  -159.990, Y  +532.100, Z    +0.000, E1  +414.924, E3 -282029.298}
SPL {X  -159.990, Y  +539.391, Z    +0.000, E1  +414.933, E3 -282040.150}
SPL {X  -159.990, Y  +546.283, Z    +0.000, E1  +414.924, E3 -282050.421}
SPL {X  -159.990, Y  +553.734, Z    +0.000, E1  +414.938, E3 -282061.508}
SPL {X  -159.990, Y  +560.657, Z    +0.000, E1  +414.914, E3 -282071.869}
SPL {X  -159.990, Y  +567.311, Z    +0.000, E1  +414.931, E3 -282081.754}
SPL {X  -159.990, Y  +577.902, Z    +0.000, E1  +414.969, E3 -282097.469}
SPL {X  -159.990, Y  +588.063, Z    +0.000, E1  +414.931, E3 -282112.660}
SPL {X  -159.990, Y  +595.273, Z    +0.000, E1  +414.928, E3 -282123.384}
SPL {X  -159.990, Y  +602.326, Z    +0.000, E1  +414.932, E3 -282133.884}
SPL {X  -159.990, Y  +609.708, Z    +0.000, E1  +414.930, E3 -282144.891}
SPL {X  -159.990, Y  +616.306, Z    +0.000, E1  +414.927, E3 -282154.704}
SPL {X  -159.990, Y  +624.320, Z    +0.000, E1  +414.952, E3 -282166.587}
SPL {X  -159.990, Y  +632.991, Z    +0.000, E1  +414.938, E3 -282179.519}
SPL {X  -159.990, Y  +639.033, Z    +0.000, E1  +414.931, E3 -282188.526}
SPL {X  -159.990, Y  +646.303, Z    +0.000, E1  +414.946, E3 -282199.314}
SPL {X  -159.990, Y  +656.335, Z    +0.000, E1  +414.969, E3 -282214.216}
SPL {X  -159.990, Y  +664.577, Z    +0.000, E1  +414.924, E3 -282226.594}
SPL {X  -159.989, Y  +672.128, Z    +0.000, E1  +414.946, E3 -282237.810}
SPL {X  -159.792, Y  +679.466, Z    +0.000, E1  +414.893, E3 -282248.968}
SPL {X  -159.330, Y  +686.016, Z    +0.000, E1  +414.837, E3 -282259.199}
SPL {X  -158.190, Y  +695.432, Z    +0.000, E1  +414.658, E3 -282274.396}
SPL {X  -157.027, Y  +702.151, Z    +0.000, E1  +414.415, E3 -282285.678}
SPL {X  -156.112, Y  +706.513, Z    +0.000, E1  +414.265, E3 -282293.112}
SPL {X  -154.917, Y  +711.470, Z    +0.000, E1  +414.052, E3 -282301.739}
SPL {X  -153.561, Y  +716.398, Z    +0.000, E1  +413.816, E3 -282310.461}
SPL {X  -151.715, Y  +722.287, Z    +0.000, E1  +413.503, E3 -282321.077}
SPL {X  -149.700, Y  +727.952, Z    +0.000, E1  +413.118, E3 -282331.551}
SPL {X  -147.376, Y  +733.767, Z    +0.000, E1  +412.706, E3 -282342.501}
SPL {X  -145.109, Y  +738.881, Z    +0.000, E1  +412.243, E3 -282352.348}
SPL {X  -142.777, Y  +743.691, Z    +0.000, E1  +411.831, E3 -282361.666}
SPL {X  -132.301, Y  +761.463, Z    +0.000, E1  +405.510, E3 -282440.951}
ENDSPLINE

SPLINE
SPL {X  -145.877, Y  +737.201, Z    +0.000, E1  +394.468, E3 -282524.062}
SPL {X  -152.550, Y  +719.721, Z    +0.000, E1  +387.728, E3 -282539.551}
SPL {X  -157.145, Y  +701.536, Z    +0.000, E1  +379.368, E3 -282549.006}
SPL {X  -159.035, Y  +688.952, Z    +0.000, E1  +372.676, E3 -282553.047}
SPL {X  -159.873, Y  +677.622, Z    +0.000, E1  +366.008, E3 -282555.119}
SPL {X  -159.990, Y  +671.638, Z    +0.000, E1  +361.925, E3 -282555.746}
SPL {X  -159.990, Y  +668.344, Z    +0.000, E1  +359.382, E3 -282555.938}
SPL {X  -159.990, Y  +664.070, Z    +0.000, E1  +354.975, E3 -282556.266}
SPL {X  -159.990, Y  +658.737, Z    +0.000, E1  +348.199, E3 -282556.972}
SPL {X  -159.990, Y  +652.023, Z    +0.000, E1  +339.551, E3 -282558.457}
SPL {X  -159.990, Y  +641.935, Z    +0.000, E1  +328.152, E3 -282561.629}
SPL {X  -159.990, Y  +605.095, Z    +0.000, E1  +310.486, E3 -282585.835}
SPL {X  -159.990, Y  +546.155, Z    +0.000, E1  +305.539, E3 -282648.594}
SPL {X  -159.990, Y  +539.348, Z    +0.000, E1  +305.531, E3 -282658.897}
SPL {X  -159.990, Y  +530.752, Z    +0.000, E1  +305.518, E3 -282671.905}
SPL {X  -159.990, Y  +522.797, Z    +0.000, E1  +305.537, E3 -282683.988}
SPL {X  -159.990, Y  +515.332, Z    +0.000, E1  +305.526, E3 -282695.277}
SPL {X  -159.990, Y  +508.047, Z    +0.000, E1  +305.531, E3 -282706.293}
SPL {X  -159.990, Y  +501.296, Z    +0.000, E1  +305.518, E3 -282716.515}
SPL {X  -159.990, Y  +487.558, Z    +0.000, E1  +304.151, E3 -282728.145}
SPL {X  -159.990, Y  +454.926, Z    +0.000, E1  +299.433, E3 -282739.585}
SPL {X  -159.990, Y  +449.697, Z    +0.000, E1  +300.191, E3 -282751.047}
SPL {X  -159.990, Y  +445.847, Z    +0.000, E1  +300.905, E3 -282760.670}
SPL {X  -159.990, Y  +439.266, Z    +0.000, E1  +301.568, E3 -282773.753}
SPL {X  -159.990, Y  +432.883, Z    +0.000, E1  +302.386, E3 -282787.444}
SPL {X  -159.990, Y  +429.044, Z    +0.000, E1  +303.109, E3 -282797.334}
SPL {X  -159.990, Y  +425.222, Z    +0.000, E1  +304.101, E3 -282809.231}
SPL {X  -159.990, Y  +418.562, Z    +0.000, E1  +304.950, E3 -282824.389}
SPL {X  -159.990, Y  +407.911, Z    +0.000, E1  +305.062, E3 -282840.980}
SPL {X  -159.990, Y  +400.284, Z    +0.000, E1  +305.103, E3 -282852.414}
SPL {X  -159.990, Y  +391.119, Z    +0.000, E1  +305.052, E3 -282866.002}
SPL {X  -159.988, Y  +381.720, Z    +0.000, E1  +305.103, E3 -282880.110}
SPL {X  -159.786, Y  +374.425, Z    +0.000, E1  +305.121, E3 -282891.158}
SPL {X  -159.015, Y  +364.863, Z    +0.000, E1  +305.220, E3 -282906.174}
SPL {X  -157.966, Y  +357.131, Z    +0.000, E1  +305.441, E3 -282918.864}
SPL {X  -156.775, Y  +350.586, Z    +0.000, E1  +305.627, E3 -282929.838}
SPL {X  -155.027, Y  +342.959, Z    +0.000, E1  +305.926, E3 -282943.011}
SPL {X  -152.882, Y  +335.340, Z    +0.000, E1  +306.305, E3 -282956.554}
SPL {X  -150.681, Y  +328.723, Z    +0.000, E1  +306.710, E3 -282968.648}
SPL {X  -148.661, Y  +323.366, Z    +0.000, E1  +307.100, E3 -282978.657}
SPL {X  -147.089, Y  +319.560, Z    +0.000, E1  +307.396, E3 -282985.873}
SPL {X  -145.161, Y  +315.232, Z    +0.000, E1  +307.745, E3 -282994.153}
SPL {X  -142.534, Y  +309.830, Z    +0.000, E1  +308.237, E3 -283004.658}
SPL {X  -132.342, Y  +292.599, Z    +0.000, E1  +315.826, E3 -283101.946}
ENDSPLINE

SPLINE
SPL {X  -151.238, Y  +330.309, Z    +0.000, E1  +330.693, E3 -283175.103}
SPL {X  -156.949, Y  +351.453, Z    +0.000, E1  +340.161, E3 -283187.264}
SPL {X  -159.024, Y  +364.945, Z    +0.000, E1  +347.297, E3 -283191.682}
SPL {X  -159.878, Y  +376.512, Z    +0.000, E1  +354.071, E3 -283193.933}
SPL {X  -159.990, Y  +383.659, Z    +0.000, E1  +358.950, E3 -283194.628}
SPL {X  -159.990, Y  +387.327, Z    +0.000, E1  +362.137, E3 -283194.861}
SPL {X  -159.990, Y  +390.622, Z    +0.000, E1  +365.876, E3 -283195.154}
SPL {X  -159.990, Y  +394.493, Z    +0.000, E1  +370.512, E3 -283195.677}
SPL {X  -159.990, Y  +401.377, Z    +0.000, E1  +379.398, E3 -283197.131}
SPL {X  -159.990, Y  +411.365, Z    +0.000, E1  +390.630, E3 -283200.340}
SPL {X  -159.990, Y  +450.467, Z    +0.000, E1  +410.183, E3 -283223.989}
SPL {X  -159.990, Y  +509.934, Z    +0.000, E1  +414.923, E3 -283286.607}
SPL {X  -159.990, Y  +516.848, Z    +0.000, E1  +414.930, E3 -283296.896}
SPL {X  -159.990, Y  +524.818, Z    +0.000, E1  +414.933, E3 -283308.767}
SPL {X  -159.990, Y  +532.100, Z    +0.000, E1  +414.924, E3 -283319.620}
SPL {X  -159.990, Y  +539.391, Z    +0.000, E1  +414.933, E3 -283330.472}
SPL {X  -159.990, Y  +546.283, Z    +0.000, E1  +414.924, E3 -283340.744}
SPL {X  -159.990, Y  +553.734, Z    +0.000, E1  +414.938, E3 -283351.831}
SPL {X  -159.990, Y  +564.956, Z    +0.000, E1  +414.973, E3 -283368.502}
SPL {X  -159.990, Y  +577.902, Z    +0.000, E1  +414.969, E3 -283387.792}
SPL {X  -159.990, Y  +588.063, Z    +0.000, E1  +414.931, E3 -283402.983}
SPL {X  -159.990, Y  +595.273, Z    +0.000, E1  +414.928, E3 -283413.706}
SPL {X  -159.990, Y  +602.326, Z    +0.000, E1  +414.932, E3 -283424.207}
SPL {X  -159.990, Y  +609.708, Z    +0.000, E1  +414.930, E3 -283435.213}
SPL {X  -159.990, Y  +618.088, Z    +0.000, E1  +414.948, E3 -283447.642}
SPL {X  -159.990, Y  +625.928, Z    +0.000, E1  +414.931, E3 -283459.338}
SPL {X  -159.990, Y  +635.803, Z    +0.000, E1  +414.980, E3 -283473.966}
SPL {X  -159.990, Y  +646.303, Z    +0.000, E1  +414.946, E3 -283489.637}
SPL {X  -159.990, Y  +656.335, Z    +0.000, E1  +414.969, E3 -283504.539}
SPL {X  -159.990, Y  +664.577, Z    +0.000, E1  +414.924, E3 -283516.916}
SPL {X  -159.989, Y  +672.128, Z    +0.000, E1  +414.946, E3 -283528.133}
SPL {X  -159.792, Y  +679.466, Z    +0.000, E1  +414.893, E3 -283539.291}
SPL {X  -159.330, Y  +686.016, Z    +0.000, E1  +414.837, E3 -283549.522}
SPL {X  -158.190, Y  +695.432, Z    +0.000, E1  +414.658, E3 -283564.718}
SPL {X  -157.027, Y  +702.151, Z    +0.000, E1  +414.415, E3 -283576.001}
SPL {X  -156.112, Y  +706.513, Z    +0.000, E1  +414.265, E3 -283583.434}
SPL {X  -154.917, Y  +711.470, Z    +0.000, E1  +414.052, E3 -283592.062}
SPL {X  -153.561, Y  +716.398, Z    +0.000, E1  +413.816, E3 -283600.783}
SPL {X  -151.715, Y  +722.287, Z    +0.000, E1  +413.503, E3 -283611.399}
SPL {X  -149.700, Y  +727.952, Z    +0.000, E1  +413.118, E3 -283621.874}
SPL {X  -147.376, Y  +733.767, Z    +0.000, E1  +412.706, E3 -283632.824}
SPL {X  -144.332, Y  +740.529, Z    +0.000, E1  +412.133, E3 -283645.814}
SPL {X  -142.065, Y  +745.081, Z    +0.000, E1  +411.654, E3 -283654.767}
SPL {X  -132.301, Y  +761.463, Z    +0.000, E1  +405.510, E3 -283731.274}
ENDSPLINE

SPLINE
SPL {X  -145.877, Y  +737.201, Z    +0.000, E1  +394.468, E3 -283814.385}
SPL {X  -152.550, Y  +719.721, Z    +0.000, E1  +387.728, E3 -283829.874}
SPL {X  -157.145, Y  +701.536, Z    +0.000, E1  +379.368, E3 -283839.329}
SPL {X  -159.035, Y  +688.952, Z    +0.000, E1  +372.676, E3 -283843.370}
SPL {X  -159.756, Y  +680.154, Z    +0.000, E1  +367.520, E3 -283845.096}
SPL {X  -159.986, Y  +672.560, Z    +0.000, E1  +362.636, E3 -283845.994}
SPL {X  -159.990, Y  +668.344, Z    +0.000, E1  +359.382, E3 -283846.260}
SPL {X  -159.990, Y  +664.070, Z    +0.000, E1  +354.975, E3 -283846.589}
SPL {X  -159.990, Y  +656.953, Z    +0.000, E1  +346.040, E3 -283847.655}
SPL {X  -159.990, Y  +644.589, Z    +0.000, E1  +330.989, E3 -283851.067}
SPL {X  -159.990, Y  +605.095, Z    +0.000, E1  +310.486, E3 -283876.158}
SPL {X  -159.990, Y  +546.155, Z    +0.000, E1  +305.539, E3 -283938.916}
SPL {X  -159.990, Y  +539.348, Z    +0.000, E1  +305.531, E3 -283949.220}
SPL {X  -159.990, Y  +530.752, Z    +0.000, E1  +305.518, E3 -283962.227}
SPL {X  -159.990, Y  +522.797, Z    +0.000, E1  +305.537, E3 -283974.310}
SPL {X  -159.990, Y  +515.332, Z    +0.000, E1  +305.526, E3 -283985.599}
SPL {X  -159.990, Y  +508.047, Z    +0.000, E1  +305.531, E3 -283996.616}
SPL {X  -159.990, Y  +499.403, Z    +0.000, E1  +305.488, E3 -284009.655}
SPL {X  -159.990, Y  +479.413, Z    +0.000, E1  +302.719, E3 -284020.801}
SPL {X  -159.990, Y  +454.926, Z    +0.000, E1  +299.433, E3 -284029.907}
SPL {X  -159.990, Y  +449.697, Z    +0.000, E1  +300.191, E3 -284041.370}
SPL {X  -159.990, Y  +445.847, Z    +0.000, E1  +300.905, E3 -284050.993}
SPL {X  -159.990, Y  +439.266, Z    +0.000, E1  +301.568, E3 -284064.076}
SPL {X  -159.990, Y  +432.883, Z    +0.000, E1  +302.386, E3 -284077.766}
SPL {X  -159.990, Y  +429.044, Z    +0.000, E1  +303.109, E3 -284087.656}
SPL {X  -159.990, Y  +425.222, Z    +0.000, E1  +304.101, E3 -284099.553}
SPL {X  -159.990, Y  +420.083, Z    +0.000, E1  +304.918, E3 -284112.129}
SPL {X  -159.990, Y  +412.567, Z    +0.000, E1  +305.072, E3 -284124.353}
SPL {X  -159.990, Y  +402.790, Z    +0.000, E1  +305.070, E3 -284138.947}
SPL {X  -159.990, Y  +391.119, Z    +0.000, E1  +305.052, E3 -284156.325}
SPL {X  -159.988, Y  +381.720, Z    +0.000, E1  +305.103, E3 -284170.432}
SPL {X  -159.786, Y  +374.425, Z    +0.000, E1  +305.121, E3 -284181.480}
SPL {X  -159.015, Y  +364.863, Z    +0.000, E1  +305.220, E3 -284196.497}
SPL {X  -157.966, Y  +357.131, Z    +0.000, E1  +305.441, E3 -284209.187}
SPL {X  -156.775, Y  +350.586, Z    +0.000, E1  +305.627, E3 -284220.161}
SPL {X  -155.027, Y  +342.959, Z    +0.000, E1  +305.926, E3 -284233.334}
SPL {X  -152.882, Y  +335.340, Z    +0.000, E1  +306.305, E3 -284246.877}
SPL {X  -150.681, Y  +328.723, Z    +0.000, E1  +306.710, E3 -284258.971}
SPL {X  -148.661, Y  +323.366, Z    +0.000, E1  +307.100, E3 -284268.980}
SPL {X  -147.089, Y  +319.560, Z    +0.000, E1  +307.396, E3 -284276.195}
SPL {X  -145.161, Y  +315.232, Z    +0.000, E1  +307.745, E3 -284284.475}
SPL {X  -142.534, Y  +309.830, Z    +0.000, E1  +308.237, E3 -284294.981}
SPL {X  -132.342, Y  +292.599, Z    +0.000, E1  +315.826, E3 -284392.269}
ENDSPLINE

SPLINE
SPL {X  -151.238, Y  +330.309, Z    +0.000, E1  +330.693, E3 -284465.425}
SPL {X  -156.949, Y  +351.453, Z    +0.000, E1  +340.161, E3 -284477.586}
SPL {X  -159.024, Y  +364.945, Z    +0.000, E1  +347.297, E3 -284482.004}
SPL {X  -159.878, Y  +376.512, Z    +0.000, E1  +354.071, E3 -284484.256}
SPL {X  -159.990, Y  +383.659, Z    +0.000, E1  +358.950, E3 -284484.950}
SPL {X  -159.990, Y  +387.327, Z    +0.000, E1  +362.137, E3 -284485.183}
SPL {X  -159.990, Y  +390.622, Z    +0.000, E1  +365.876, E3 -284485.476}
SPL {X  -159.990, Y  +394.493, Z    +0.000, E1  +370.512, E3 -284485.999}
SPL {X  -159.990, Y  +401.377, Z    +0.000, E1  +379.398, E3 -284487.454}
SPL {X  -159.990, Y  +411.365, Z    +0.000, E1  +390.630, E3 -284490.662}
SPL {X  -159.990, Y  +450.467, Z    +0.000, E1  +410.183, E3 -284514.311}
SPL {X  -159.990, Y  +509.934, Z    +0.000, E1  +414.923, E3 -284576.930}
SPL {X  -159.990, Y  +516.848, Z    +0.000, E1  +414.930, E3 -284587.218}
SPL {X  -159.990, Y  +524.818, Z    +0.000, E1  +414.933, E3 -284599.090}
SPL {X  -159.990, Y  +532.100, Z    +0.000, E1  +414.924, E3 -284609.943}
SPL {X  -159.990, Y  +539.391, Z    +0.000, E1  +414.933, E3 -284620.795}
SPL {X  -159.990, Y  +546.283, Z    +0.000, E1  +414.924, E3 -284631.067}
SPL {X  -159.990, Y  +553.734, Z    +0.000, E1  +414.938, E3 -284642.153}
SPL {X  -159.990, Y  +564.956, Z    +0.000, E1  +414.973, E3 -284658.825}
SPL {X  -159.990, Y  +577.902, Z    +0.000, E1  +414.969, E3 -284678.114}
SPL {X  -159.990, Y  +588.063, Z    +0.000, E1  +414.931, E3 -284693.305}
SPL {X  -159.990, Y  +595.273, Z    +0.000, E1  +414.928, E3 -284704.029}
SPL {X  -159.990, Y  +602.326, Z    +0.000, E1  +414.932, E3 -284714.529}
SPL {X  -159.990, Y  +609.708, Z    +0.000, E1  +414.930, E3 -284725.536}
SPL {X  -159.990, Y  +618.088, Z    +0.000, E1  +414.948, E3 -284737.965}
SPL {X  -159.990, Y  +625.928, Z    +0.000, E1  +414.931, E3 -284749.661}
SPL {X  -159.990, Y  +635.803, Z    +0.000, E1  +414.980, E3 -284764.289}
SPL {X  -159.990, Y  +646.303, Z    +0.000, E1  +414.946, E3 -284779.959}
SPL {X  -159.990, Y  +653.312, Z    +0.000, E1  +414.932, E3 -284790.411}
SPL {X  -159.990, Y  +658.943, Z    +0.000, E1  +414.931, E3 -284798.809}
SPL {X  -159.990, Y  +667.151, Z    +0.000, E1  +414.954, E3 -284811.028}
SPL {X  -159.885, Y  +677.285, Z    +0.000, E1  +414.936, E3 -284826.223}
SPL {X  -159.482, Y  +684.244, Z    +0.000, E1  +414.840, E3 -284837.075}
SPL {X  -158.805, Y  +690.934, Z    +0.000, E1  +414.742, E3 -284847.724}
SPL {X  -157.890, Y  +697.337, Z    +0.000, E1  +414.571, E3 -284858.246}
SPL {X  -156.492, Y  +704.774, Z    +0.000, E1  +414.365, E3 -284870.725}
SPL {X  -154.917, Y  +711.470, Z    +0.000, E1  +414.052, E3 -284882.385}
SPL {X  -153.561, Y  +716.398, Z    +0.000, E1  +413.816, E3 -284891.106}
SPL {X  -151.715, Y  +722.287, Z    +0.000, E1  +413.503, E3 -284901.722}
SPL {X  -148.967, Y  +729.859, Z    +0.000, E1  +413.026, E3 -284915.714}
SPL {X  -145.862, Y  +737.236, Z    +0.000, E1  +412.427, E3 -284929.768}
SPL {X  -142.777, Y  +743.691, Z    +0.000, E1  +411.831, E3 -284942.312}
SPL {X  -132.301, Y  +761.463, Z    +0.000, E1  +405.510, E3 -285021.597}
ENDSPLINE

SPLINE
SPL {X  -145.877, Y  +737.201, Z    +0.000, E1  +394.468, E3 -285104.707}
SPL {X  -152.550, Y  +719.721, Z    +0.000, E1  +387.728, E3 -285120.197}
SPL {X  -157.145, Y  +701.536, Z    +0.000, E1  +379.368, E3 -285129.651}
SPL {X  -159.035, Y  +688.952, Z    +0.000, E1  +372.676, E3 -285133.692}
SPL {X  -159.756, Y  +680.154, Z    +0.000, E1  +367.520, E3 -285135.419}
SPL {X  -159.986, Y  +672.560, Z    +0.000, E1  +362.636, E3 -285136.317}
SPL {X  -159.990, Y  +668.344, Z    +0.000, E1  +359.382, E3 -285136.583}
SPL {X  -159.990, Y  +664.070, Z    +0.000, E1  +354.975, E3 -285136.911}
SPL {X  -159.990, Y  +656.953, Z    +0.000, E1  +346.040, E3 -285137.978}
SPL {X  -159.990, Y  +644.589, Z    +0.000, E1  +330.989, E3 -285141.389}
SPL {X  -159.990, Y  +605.095, Z    +0.000, E1  +310.486, E3 -285166.480}
SPL {X  -159.990, Y  +546.155, Z    +0.000, E1  +305.539, E3 -285229.239}
SPL {X  -159.990, Y  +539.348, Z    +0.000, E1  +305.531, E3 -285239.543}
SPL {X  -159.990, Y  +530.752, Z    +0.000, E1  +305.518, E3 -285252.550}
SPL {X  -159.990, Y  +522.797, Z    +0.000, E1  +305.537, E3 -285264.633}
SPL {X  -159.990, Y  +515.332, Z    +0.000, E1  +305.526, E3 -285275.922}
SPL {X  -159.990, Y  +508.047, Z    +0.000, E1  +305.531, E3 -285286.939}
SPL {X  -159.990, Y  +501.296, Z    +0.000, E1  +305.518, E3 -285297.160}
SPL {X  -159.990, Y  +487.558, Z    +0.000, E1  +304.151, E3 -285308.791}
SPL {X  -159.990, Y  +454.926, Z    +0.000, E1  +299.433, E3 -285320.230}
SPL {X  -159.990, Y  +449.697, Z    +0.000, E1  +300.191, E3 -285331.692}
SPL {X  -159.990, Y  +445.847, Z    +0.000, E1  +300.905, E3 -285341.315}
SPL {X  -159.990, Y  +439.266, Z    +0.000, E1  +301.568, E3 -285354.398}
SPL {X  -159.990, Y  +432.883, Z    +0.000, E1  +302.386, E3 -285368.089}
SPL {X  -159.990, Y  +429.044, Z    +0.000, E1  +303.109, E3 -285377.979}
SPL {X  -159.990, Y  +425.222, Z    +0.000, E1  +304.101, E3 -285389.876}
SPL {X  -159.990, Y  +418.562, Z    +0.000, E1  +304.950, E3 -285405.034}
SPL {X  -159.990, Y  +407.911, Z    +0.000, E1  +305.062, E3 -285421.625}
SPL {X  -159.990, Y  +400.284, Z    +0.000, E1  +305.103, E3 -285433.059}
SPL {X  -159.990, Y  +391.119, Z    +0.000, E1  +305.052, E3 -285446.647}
SPL {X  -159.988, Y  +381.720, Z    +0.000, E1  +305.103, E3 -285460.755}
SPL {X  -159.786, Y  +374.425, Z    +0.000, E1  +305.121, E3 -285471.803}
SPL {X  -159.015, Y  +364.863, Z    +0.000, E1  +305.220, E3 -285486.819}
SPL {X  -157.966, Y  +357.131, Z    +0.000, E1  +305.441, E3 -285499.510}
SPL {X  -156.775, Y  +350.586, Z    +0.000, E1  +305.627, E3 -285510.483}
SPL {X  -155.027, Y  +342.959, Z    +0.000, E1  +305.926, E3 -285523.656}
SPL {X  -152.882, Y  +335.340, Z    +0.000, E1  +306.305, E3 -285537.199}
SPL {X  -150.681, Y  +328.723, Z    +0.000, E1  +306.710, E3 -285549.293}
SPL {X  -148.661, Y  +323.366, Z    +0.000, E1  +307.100, E3 -285559.303}
SPL {X  -147.089, Y  +319.560, Z    +0.000, E1  +307.396, E3 -285566.518}
SPL {X  -145.161, Y  +315.232, Z    +0.000, E1  +307.745, E3 -285574.798}
SPL {X  -142.534, Y  +309.830, Z    +0.000, E1  +308.237, E3 -285585.303}
SPL {X  -132.342, Y  +292.599, Z    +0.000, E1  +315.826, E3 -285682.591}
ENDSPLINE

SPLINE
SPL {X  -151.238, Y  +330.309, Z    +0.000, E1  +330.693, E3 -285755.748}
SPL {X  -156.949, Y  +351.453, Z    +0.000, E1  +340.161, E3 -285767.909}
SPL {X  -159.024, Y  +364.945, Z    +0.000, E1  +347.297, E3 -285772.327}
SPL {X  -159.758, Y  +373.891, Z    +0.000, E1  +352.513, E3 -285774.215}
SPL {X  -159.985, Y  +381.208, Z    +0.000, E1  +357.184, E3 -285775.098}
SPL {X  -159.990, Y  +384.493, Z    +0.000, E1  +359.676, E3 -285775.323}
SPL {X  -159.990, Y  +387.327, Z    +0.000, E1  +362.137, E3 -285775.506}
SPL {X  -159.990, Y  +392.053, Z    +0.000, E1  +367.477, E3 -285775.971}
SPL {X  -159.990, Y  +396.158, Z    +0.000, E1  +372.775, E3 -285776.596}
SPL {X  -159.990, Y  +401.377, Z    +0.000, E1  +379.398, E3 -285777.776}
SPL {X  -159.990, Y  +411.365, Z    +0.000, E1  +390.630, E3 -285780.985}
SPL {X  -159.990, Y  +450.467, Z    +0.000, E1  +410.183, E3 -285804.634}
SPL {X  -159.990, Y  +509.934, Z    +0.000, E1  +414.923, E3 -285867.253}
SPL {X  -159.990, Y  +516.848, Z    +0.000, E1  +414.930, E3 -285877.541}
SPL {X  -159.990, Y  +524.818, Z    +0.000, E1  +414.933, E3 -285889.413}
SPL {X  -159.990, Y  +532.100, Z    +0.000, E1  +414.924, E3 -285900.266}
SPL {X  -159.990, Y  +539.391, Z    +0.000, E1  +414.933, E3 -285911.118}
SPL {X  -159.990, Y  +546.283, Z    +0.000, E1  +414.924, E3 -285921.389}
SPL {X  -159.990, Y  +553.734, Z    +0.000, E1  +414.938, E3 -285932.476}
SPL {X  -159.990, Y  +564.956, Z    +0.000, E1  +414.973, E3 -285949.147}
SPL {X  -159.990, Y  +577.902, Z    +0.000, E1  +414.969, E3 -285968.437}
SPL {X  -159.990, Y  +588.063, Z    +0.000, E1  +414.931, E3 -285983.628}
SPL {X  -159.990, Y  +595.273, Z    +0.000, E1  +414.928, E3 -285994.351}
SPL {X  -159.990, Y  +602.326, Z    +0.000, E1  +414.932, E3 -286004.852}
SPL {X  -159.990, Y  +609.708, Z    +0.000, E1  +414.930, E3 -286015.858}
SPL {X  -159.990, Y  +618.088, Z    +0.000, E1  +414.948, E3 -286028.287}
SPL {X  -159.990, Y  +625.928, Z    +0.000, E1  +414.931, E3 -286039.983}
SPL {X  -159.990, Y  +632.991, Z    +0.000, E1  +414.938, E3 -286050.486}
SPL {X  -159.990, Y  +639.033, Z    +0.000, E1  +414.931, E3 -286059.494}
SPL {X  -159.990, Y  +646.303, Z    +0.000, E1  +414.946, E3 -286070.282}
SPL {X  -159.990, Y  +656.335, Z    +0.000, E1  +414.969, E3 -286085.184}
SPL {X  -159.990, Y  +664.577, Z    +0.000, E1  +414.924, E3 -286097.562}
SPL {X  -159.989, Y  +672.128, Z    +0.000, E1  +414.946, E3 -286108.778}
SPL {X  -159.636, Y  +682.136, Z    +0.000, E1  +414.901, E3 -286124.036}
SPL {X  -158.805, Y  +690.934, Z    +0.000, E1  +414.742, E3 -286138.047}
SPL {X  -157.890, Y  +697.337, Z    +0.000, E1  +414.571, E3 -286148.568}
SPL {X  -156.492, Y  +704.774, Z    +0.000, E1  +414.365, E3 -286161.047}
SPL {X  -154.917, Y  +711.470, Z    +0.000, E1  +414.052, E3 -286172.707}
SPL {X  -153.204, Y  +717.603, Z    +0.000, E1  +413.775, E3 -286183.553}
SPL {X  -151.355, Y  +723.351, Z    +0.000, E1  +413.415, E3 -286194.025}
SPL {X  -148.967, Y  +729.859, Z    +0.000, E1  +413.026, E3 -286206.037}
SPL {X  -145.862, Y  +737.236, Z    +0.000, E1  +412.427, E3 -286220.091}
SPL {X  -142.777, Y  +743.691, Z    +0.000, E1  +411.831, E3 -286232.634}
SPL {X  -132.301, Y  +761.463, Z    +0.000, E1  +405.510, E3 -286311.919}
ENDSPLINE

